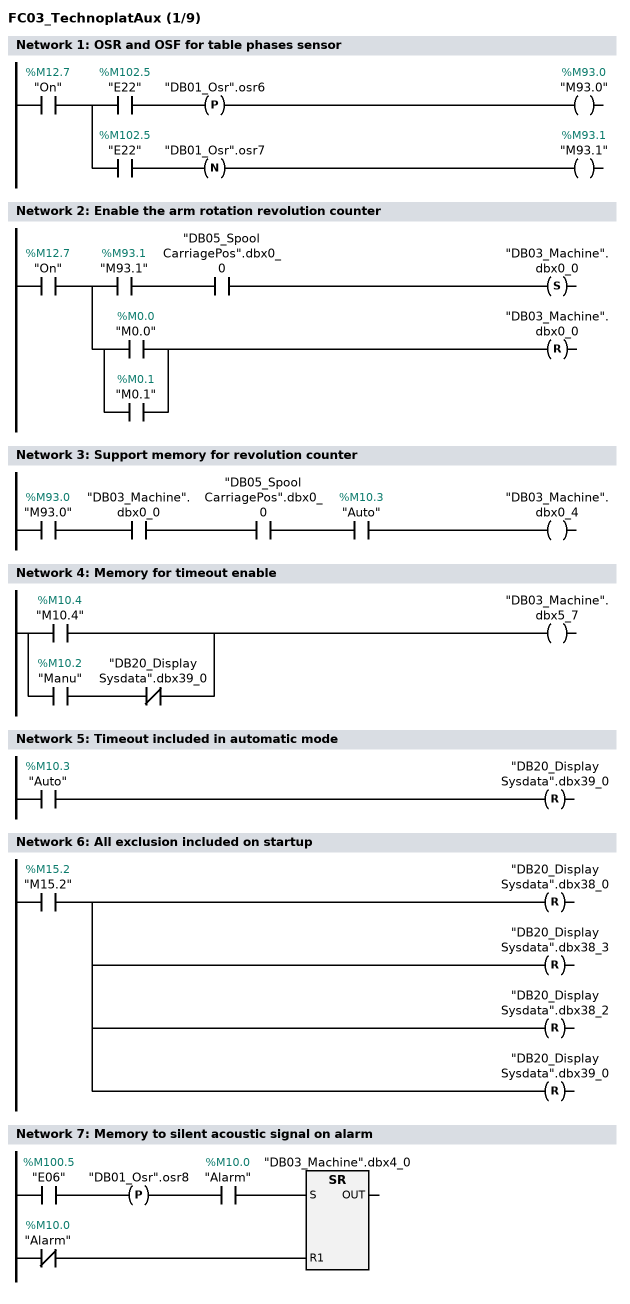
   RUNG wire#powerrail
      Contact( "On" )
      wire#w1
      Contact( "E22" )
      P_Trig( "DB01_Osr".osr6 )
      Coil( "M93.0" )
   END_RUNG
   RUNG wire#w1
      Contact( "E22" )
      N_Trig( "DB01_Osr".osr7 )
      Coil( "M93.1" )
   END_RUNG
   // the same network as SCL:
   #_w1 := "On" AND "E22";
   #_w2 := #_w1 AND NOT "DB01_Osr".osr6;   // rising edge
   "DB01_Osr".osr6 := #_w1;
   "M93.0" := #_w2;
   #_w3 := "On" AND "E22";
   #_w4 := NOT #_w3 AND "DB01_Osr".osr7;   // falling edge
   "DB01_Osr".osr7 := #_w3;
   "M93.1" := #_w4;
END_REGION

REGION Network 2: Enable the arm rotation revolution counter
   RUNG wire#powerrail
      Contact( "On" )
      wire#w1
      Contact( "M93.1" )
      Contact( "DB05_SpoolCarriagePos".dbx0_0 )
      S_Coil( "DB03_Machine".dbx0_0 )
   END_RUNG
   RUNG wire#w1
      Contact( "M0.0" )
      wire#w2
      R_Coil( "DB03_Machine".dbx0_0 )
   END_RUNG
   RUNG wire#w1
      Contact( "M0.1" )
   END_RUNG wire#w2
   // the same network as SCL:
   IF "On" AND "M93.1" AND "DB05_SpoolCarriagePos".dbx0_0 THEN "DB03_Machine".dbx0_0 := TRUE; END_IF;
   IF "On" AND ("M0.0" OR "M0.1") THEN "DB03_Machine".dbx0_0 := FALSE; END_IF;
END_REGION

REGION Network 3: Support memory for revolution counter
   RUNG wire#powerrail
      Contact( "M93.0" )
      Contact( "DB03_Machine".dbx0_0 )
      Contact( "DB05_SpoolCarriagePos".dbx0_0 )
      Contact( "Auto" )
      Coil( "DB03_Machine".dbx0_4 )
   END_RUNG
   // the same network as SCL:
   "DB03_Machine".dbx0_4 := "M93.0" AND "DB03_Machine".dbx0_0 AND "DB05_SpoolCarriagePos".dbx0_0 AND "Auto";
END_REGION

REGION Network 4: Memory for timeout enable
   RUNG wire#powerrail
      Contact( "M10.4" )
      wire#w1
      Coil( "DB03_Machine".dbx5_7 )
   END_RUNG
   RUNG wire#powerrail
      Contact( "Manu" )
      I_Contact( "DB20_DisplaySysdata".dbx39_0 )
   END_RUNG wire#w1
   // the same network as SCL:
   "DB03_Machine".dbx5_7 := "M10.4" OR ("Manu" AND NOT "DB20_DisplaySysdata".dbx39_0);
END_REGION

REGION Network 5: Timeout included in automatic mode
   RUNG wire#powerrail
      Contact( "Auto" )
      R_Coil( "DB20_DisplaySysdata".dbx39_0 )
   END_RUNG
   // the same network as SCL:
   IF "Auto" THEN "DB20_DisplaySysdata".dbx39_0 := FALSE; END_IF;
END_REGION

REGION Network 6: All exclusion included on startup
   RUNG wire#powerrail
      Contact( "M15.2" )
      wire#w1
      R_Coil( "DB20_DisplaySysdata".dbx38_0 )
   END_RUNG
   RUNG wire#w1
      R_Coil( "DB20_DisplaySysdata".dbx38_3 )
   END_RUNG
   RUNG wire#w1
      R_Coil( "DB20_DisplaySysdata".dbx38_2 )
   END_RUNG
   RUNG wire#w1
      R_Coil( "DB20_DisplaySysdata".dbx39_0 )
   END_RUNG
   // the same network as SCL:
   IF "M15.2" THEN
       "DB20_DisplaySysdata".dbx38_0 := FALSE;
       "DB20_DisplaySysdata".dbx38_3 := FALSE;
       "DB20_DisplaySysdata".dbx38_2 := FALSE;
       "DB20_DisplaySysdata".dbx39_0 := FALSE;
   END_IF;
END_REGION

REGION Network 7: Memory to silent acoustic signal on alarm
   RUNG wire#powerrail
      Contact( "E06" )
      P_Trig( "DB01_Osr".osr8 )
      Contact( "Alarm" )
      S_SR(operand := "DB03_Machine".dbx4_0, r1 := wire#w1)
   END_RUNG
   RUNG wire#powerrail
      I_Contact( "Alarm" )
   END_RUNG wire#w1
   // the same network as SCL:
   #_w1 := "E06" AND NOT "DB01_Osr".osr8;   // rising edge
   "DB01_Osr".osr8 := "E06";
   IF #_w1 AND "Alarm" THEN
       "DB03_Machine".dbx4_0 := TRUE;   // SR flip-flop
   END_IF;
   IF NOT "Alarm" THEN "DB03_Machine".dbx4_0 := FALSE; END_IF;
END_REGION

REGION Network 8: All units are ready for automatic cycle
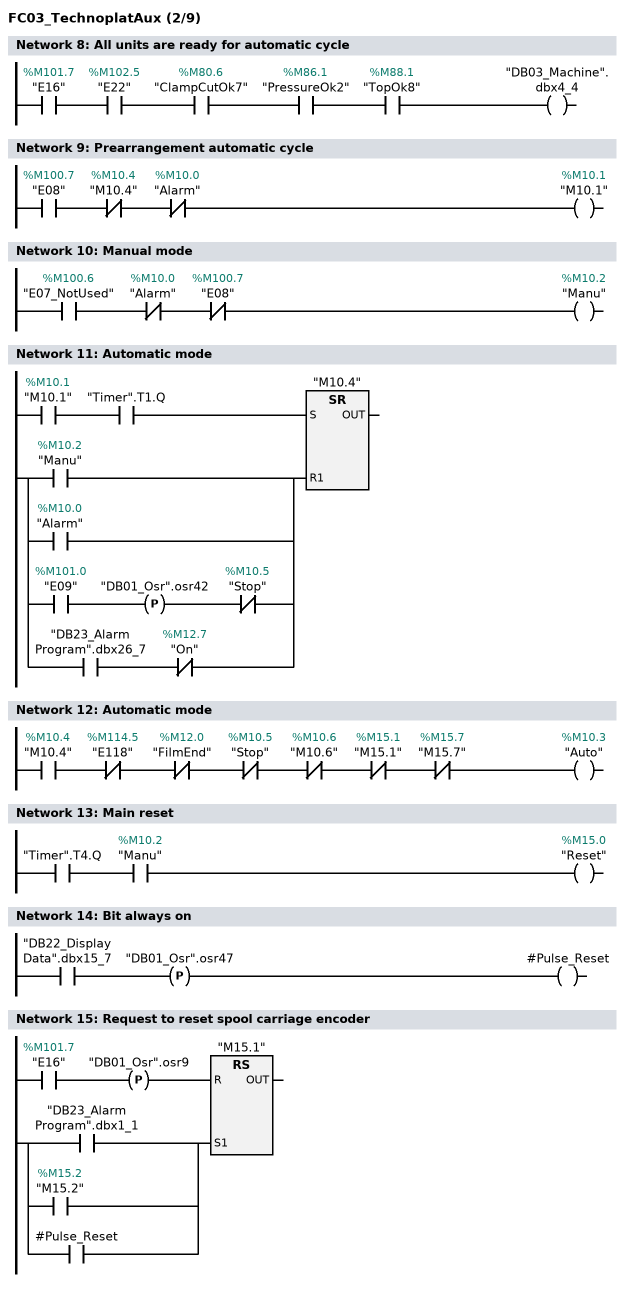
   RUNG wire#powerrail
      Contact( "E16" )
      Contact( "E22" )
      Contact( "ClampCutOk7" )
      Contact( "PressureOk2" )
      Contact( "TopOk8" )
      Coil( "DB03_Machine".dbx4_4 )
   END_RUNG
   // the same network as SCL:
   "DB03_Machine".dbx4_4 := "E16" AND "E22" AND "ClampCutOk7" AND "PressureOk2" AND "TopOk8";
END_REGION

REGION Network 9: Prearrangement automatic cycle
   RUNG wire#powerrail
      Contact( "E08" )
      I_Contact( "M10.4" )
      I_Contact( "Alarm" )
      Coil( "M10.1" )
   END_RUNG
   // the same network as SCL:
   "M10.1" := "E08" AND NOT "M10.4" AND NOT "Alarm";
END_REGION

REGION Network 10: Manual mode
   RUNG wire#powerrail
      Contact( "E07_NotUsed" )
      I_Contact( "Alarm" )
      I_Contact( "E08" )
      Coil( "Manu" )
   END_RUNG
   // the same network as SCL:
   "Manu" := "E07_NotUsed" AND NOT "Alarm" AND NOT "E08";
END_REGION

REGION Network 11: Automatic mode
   RUNG wire#powerrail
      Contact( "M10.1" )
      Contact( "Timer".T1.Q )
      S_SR(operand := "M10.4", r1 := wire#w1)
   END_RUNG
   RUNG wire#powerrail
      Contact( "Manu" )
   END_RUNG wire#w1
   RUNG wire#powerrail
      Contact( "Alarm" )
   END_RUNG wire#w1
   RUNG wire#powerrail
      Contact( "E09" )
      P_Trig( "DB01_Osr".osr42 )
      I_Contact( "Stop" )
   END_RUNG wire#w1
   RUNG wire#powerrail
      Contact( "DB23_AlarmProgram".dbx26_7 )
      I_Contact( "On" )
   END_RUNG wire#w1
   // the same network as SCL:
   #_w1 := "E09" AND NOT "DB01_Osr".osr42;   // rising edge
   "DB01_Osr".osr42 := "E09";
   IF "M10.1" AND "Timer".T1.Q THEN
       "M10.4" := TRUE;   // SR flip-flop
   END_IF;
   IF "Manu" OR "Alarm" OR (#_w1 AND NOT "Stop") OR ("DB23_AlarmProgram".dbx26_7 AND NOT "On") THEN
       "M10.4" := FALSE;
   END_IF;
END_REGION

REGION Network 12: Automatic mode
   RUNG wire#powerrail
      Contact( "M10.4" )
      I_Contact( "E118" )
      I_Contact( "FilmEnd" )
      I_Contact( "Stop" )
      I_Contact( "M10.6" )
      I_Contact( "M15.1" )
      I_Contact( "M15.7" )
      Coil( "Auto" )
   END_RUNG
   // the same network as SCL:
   "Auto" := "M10.4" AND NOT "E118" AND NOT "FilmEnd" AND NOT "Stop" AND NOT "M10.6" AND NOT "M15.1" AND NOT "M15.7";
END_REGION

REGION Network 13: Main reset
   RUNG wire#powerrail
      Contact( "Timer".T4.Q )
      Contact( "Manu" )
      Coil( "Reset" )
   END_RUNG
   // the same network as SCL:
   "Reset" := "Timer".T4.Q AND "Manu";
END_REGION

REGION Network 14: Bit always on
   RUNG wire#powerrail
      Contact( "DB22_DisplayData".dbx15_7 )
      P_Trig( "DB01_Osr".osr47 )
      Coil( #Pulse_Reset )
   END_RUNG
   // the same network as SCL:
   #_w1 := "DB22_DisplayData".dbx15_7 AND NOT "DB01_Osr".osr47;   // rising edge
   "DB01_Osr".osr47 := "DB22_DisplayData".dbx15_7;
   #Pulse_Reset := #_w1;
END_REGION

REGION Network 15: Request to reset spool carriage encoder
   RUNG wire#powerrail
      Contact( "E16" )
      P_Trig( "DB01_Osr".osr9 )
      S_RS(operand := "M15.1", s1 := wire#w1)
   END_RUNG
   RUNG wire#powerrail
      Contact( "DB23_AlarmProgram".dbx1_1 )
   END_RUNG wire#w1
   RUNG wire#powerrail
      Contact( "M15.2" )
   END_RUNG wire#w1
   RUNG wire#powerrail
      Contact( #Pulse_Reset )
   END_RUNG wire#w1
   // the same network as SCL:
   #_w1 := "E16" AND NOT "DB01_Osr".osr9;   // rising edge
   "DB01_Osr".osr9 := "E16";
   IF #_w1 THEN
       "M15.1" := FALSE;   // RS flip-flop
   END_IF;
   IF "DB23_AlarmProgram".dbx1_1 OR "M15.2" OR #Pulse_Reset THEN "M15.1" := TRUE; END_IF;
END_REGION

REGION Network 16: Request to reset table rotation encoder
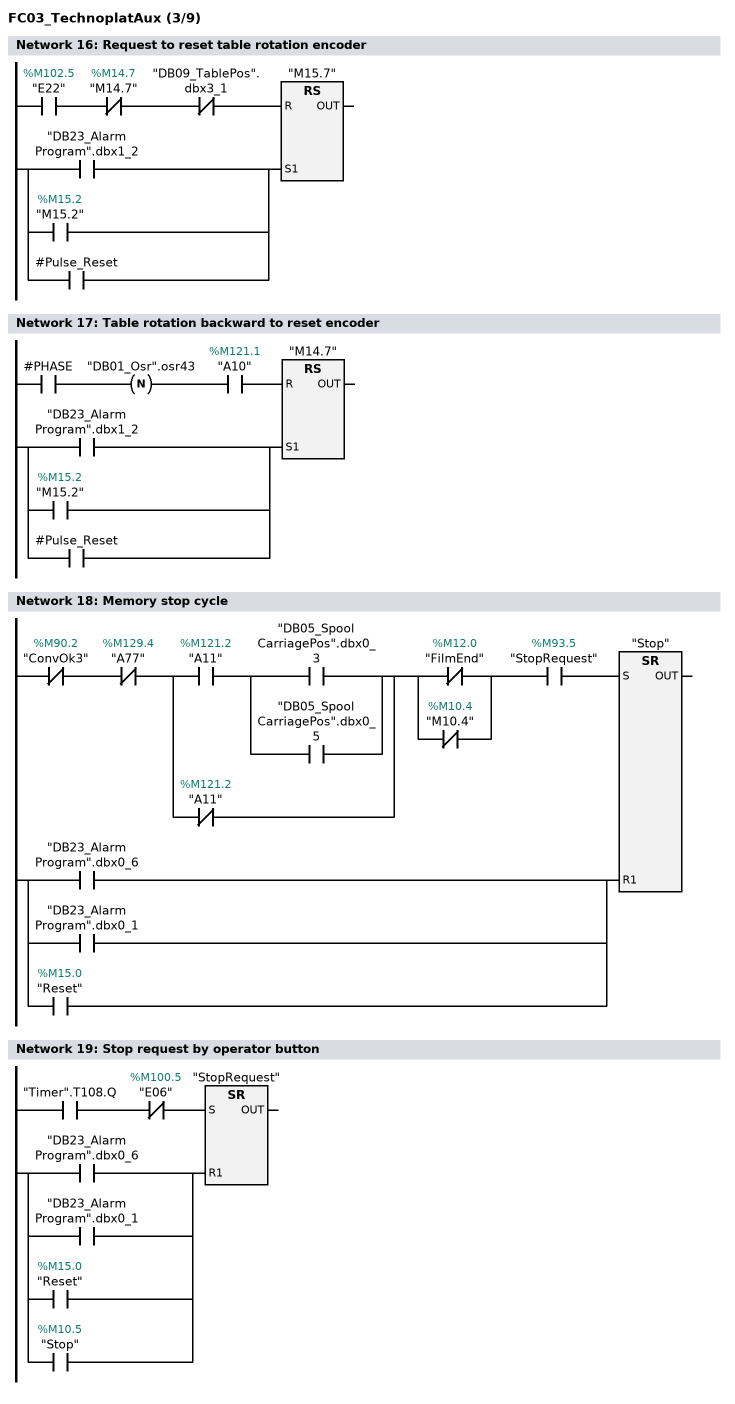
   RUNG wire#powerrail
      Contact( "E22" )
      I_Contact( "M14.7" )
      I_Contact( "DB09_TablePos".dbx3_1 )
      S_RS(operand := "M15.7", s1 := wire#w1)
   END_RUNG
   RUNG wire#powerrail
      Contact( "DB23_AlarmProgram".dbx1_2 )
   END_RUNG wire#w1
   RUNG wire#powerrail
      Contact( "M15.2" )
   END_RUNG wire#w1
   RUNG wire#powerrail
      Contact( #Pulse_Reset )
   END_RUNG wire#w1
   // the same network as SCL:
   IF "E22" AND NOT "M14.7" AND NOT "DB09_TablePos".dbx3_1 THEN
       "M15.7" := FALSE;   // RS flip-flop
   END_IF;
   IF "DB23_AlarmProgram".dbx1_2 OR "M15.2" OR #Pulse_Reset THEN "M15.7" := TRUE; END_IF;
END_REGION

REGION Network 17: Table rotation backward to reset encoder
   RUNG wire#powerrail
      Contact( #PHASE )
      N_Trig( "DB01_Osr".osr43 )
      Contact( "A10" )
      S_RS(operand := "M14.7", s1 := wire#w1)
   END_RUNG
   RUNG wire#powerrail
      Contact( "DB23_AlarmProgram".dbx1_2 )
   END_RUNG wire#w1
   RUNG wire#powerrail
      Contact( "M15.2" )
   END_RUNG wire#w1
   RUNG wire#powerrail
      Contact( #Pulse_Reset )
   END_RUNG wire#w1
   // the same network as SCL:
   #_w1 := NOT #PHASE AND "DB01_Osr".osr43;   // falling edge
   "DB01_Osr".osr43 := #PHASE;
   IF #_w1 AND "A10" THEN
       "M14.7" := FALSE;   // RS flip-flop
   END_IF;
   IF "DB23_AlarmProgram".dbx1_2 OR "M15.2" OR #Pulse_Reset THEN "M14.7" := TRUE; END_IF;
END_REGION

REGION Network 18: Memory stop cycle
   RUNG wire#powerrail
      I_Contact( "ConvOk3" )
      I_Contact( "A77" )
      wire#w1
      Contact( "A11" )
      wire#w2
      Contact( "DB05_SpoolCarriagePos".dbx0_3 )
      wire#w3
      I_Contact( "FilmEnd" )
      wire#w4
      Contact( "StopRequest" )
      S_SR(operand := "Stop", r1 := wire#w5)
   END_RUNG
   RUNG wire#w2
      Contact( "DB05_SpoolCarriagePos".dbx0_5 )
   END_RUNG wire#w3
   RUNG wire#w1
      I_Contact( "A11" )
   END_RUNG wire#w3
   RUNG wire#w3
      I_Contact( "M10.4" )
   END_RUNG wire#w4
   RUNG wire#powerrail
      Contact( "DB23_AlarmProgram".dbx0_6 )
   END_RUNG wire#w5
   RUNG wire#powerrail
      Contact( "DB23_AlarmProgram".dbx0_1 )
   END_RUNG wire#w5
   RUNG wire#powerrail
      Contact( "Reset" )
   END_RUNG wire#w5
   // the same network as SCL:
   IF NOT "ConvOk3" AND NOT "A77" AND (("A11" AND ("DB05_SpoolCarriagePos".dbx0_3 OR "DB05_SpoolCarriagePos".dbx0_5)) OR NOT "A11") AND (NOT "FilmEnd" OR NOT "M10.4") AND "StopRequest" THEN
       "Stop" := TRUE;   // SR flip-flop
   END_IF;
   IF "DB23_AlarmProgram".dbx0_6 OR "DB23_AlarmProgram".dbx0_1 OR "Reset" THEN "Stop" := FALSE; END_IF;
END_REGION

REGION Network 19: Stop request by operator button
   RUNG wire#powerrail
      Contact( "Timer".T108.Q )
      I_Contact( "E06" )
      S_SR(operand := "StopRequest", r1 := wire#w1)
   END_RUNG
   RUNG wire#powerrail
      Contact( "DB23_AlarmProgram".dbx0_6 )
   END_RUNG wire#w1
   RUNG wire#powerrail
      Contact( "DB23_AlarmProgram".dbx0_1 )
   END_RUNG wire#w1
   RUNG wire#powerrail
      Contact( "Reset" )
   END_RUNG wire#w1
   RUNG wire#powerrail
      Contact( "Stop" )
   END_RUNG wire#w1
   // the same network as SCL:
   IF "Timer".T108.Q AND NOT "E06" THEN
       "StopRequest" := TRUE;   // SR flip-flop
   END_IF;
   IF "DB23_AlarmProgram".dbx0_6 OR "DB23_AlarmProgram".dbx0_1 OR "Reset" OR "Stop" THEN
       "StopRequest" := FALSE;
   END_IF;
END_REGION

REGION Network 20: Memory to stop cycle for door open request
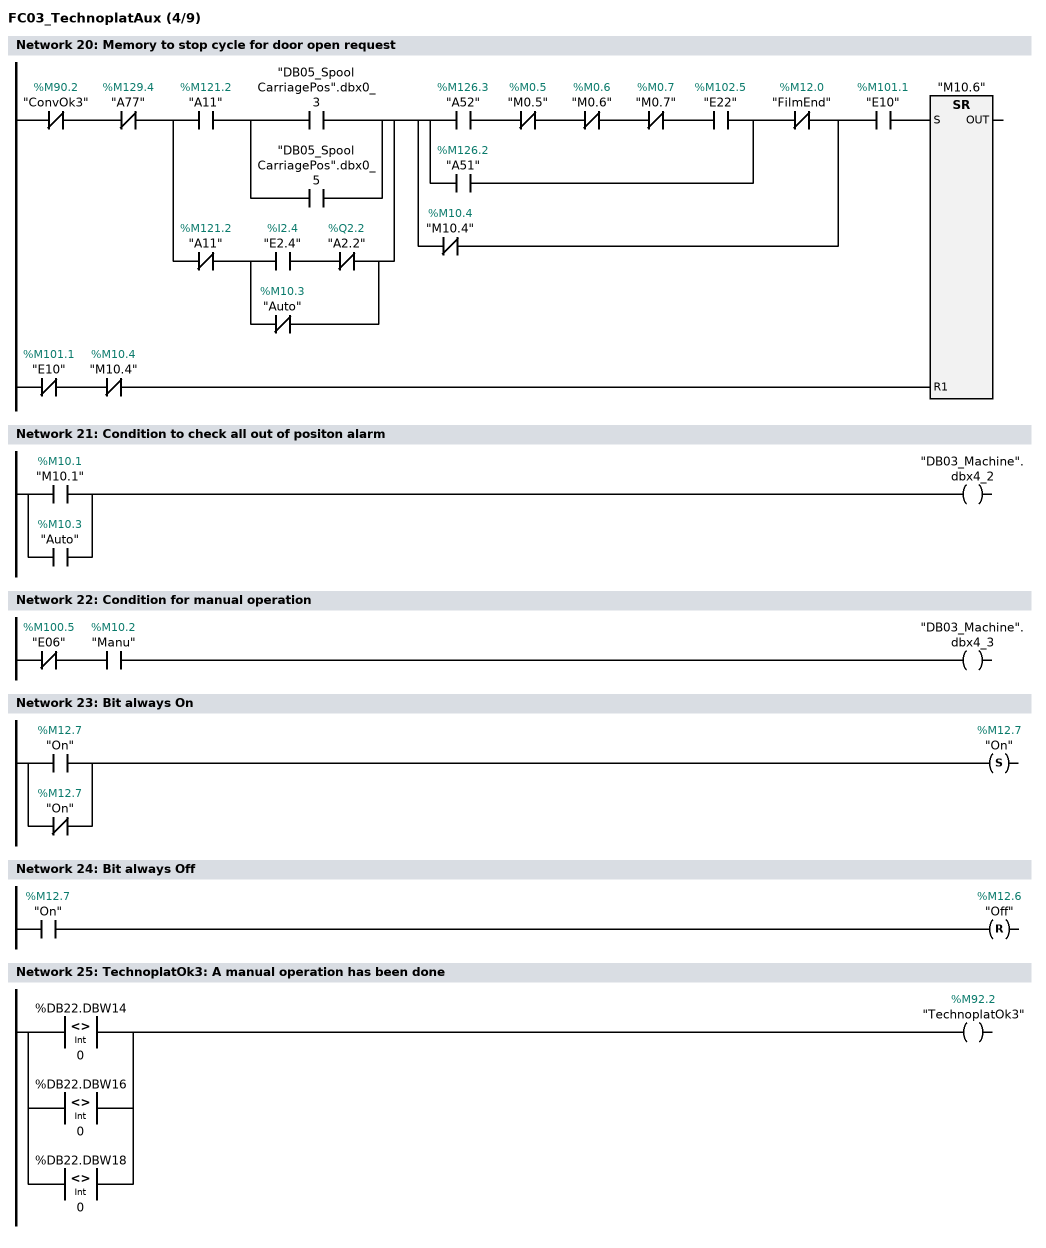
   RUNG wire#powerrail
      I_Contact( "ConvOk3" )
      I_Contact( "A77" )
      wire#w1
      Contact( "A11" )
      wire#w2
      Contact( "DB05_SpoolCarriagePos".dbx0_3 )
      wire#w3
      Contact( "A52" )
      I_Contact( "M0.5" )
      I_Contact( "M0.6" )
      I_Contact( "M0.7" )
      Contact( "E22" )
      wire#w5
      I_Contact( "FilmEnd" )
      wire#w6
      Contact( "E10" )
      S_SR(operand := "M10.6", r1 := wire#w7)
   END_RUNG
   RUNG wire#w2
      Contact( "DB05_SpoolCarriagePos".dbx0_5 )
   END_RUNG wire#w3
   RUNG wire#w1
      I_Contact( "A11" )
      wire#w4
      Contact( "E2.4" )
      I_Contact( "A2.2" )
   END_RUNG wire#w3
   RUNG wire#w4
      I_Contact( "Auto" )
   END_RUNG wire#w3
   RUNG wire#w3
      Contact( "A51" )
   END_RUNG wire#w5
   RUNG wire#w3
      I_Contact( "M10.4" )
   END_RUNG wire#w6
   RUNG wire#powerrail
      I_Contact( "E10" )
      I_Contact( "M10.4" )
   END_RUNG wire#w7
   // the same network as SCL:
   IF NOT "ConvOk3" AND NOT "A77" AND (("A11" AND ("DB05_SpoolCarriagePos".dbx0_3 OR "DB05_SpoolCarriagePos".dbx0_5)) OR (NOT "A11" AND (("E2.4" AND NOT "A2.2") OR NOT "Auto"))) AND (((("A52" AND NOT "M0.5" AND NOT "M0.6" AND NOT "M0.7" AND "E22") OR "A51") AND NOT "FilmEnd") OR NOT "M10.4") AND "E10" THEN
       "M10.6" := TRUE;   // SR flip-flop
   END_IF;
   IF NOT "E10" AND NOT "M10.4" THEN "M10.6" := FALSE; END_IF;
END_REGION

REGION Network 21: Condition to check all out of positon alarm
   RUNG wire#powerrail
      Contact( "M10.1" )
      wire#w1
      Coil( "DB03_Machine".dbx4_2 )
   END_RUNG
   RUNG wire#powerrail
      Contact( "Auto" )
   END_RUNG wire#w1
   // the same network as SCL:
   "DB03_Machine".dbx4_2 := "M10.1" OR "Auto";
END_REGION

REGION Network 22: Condition for manual operation
   RUNG wire#powerrail
      I_Contact( "E06" )
      Contact( "Manu" )
      Coil( "DB03_Machine".dbx4_3 )
   END_RUNG
   // the same network as SCL:
   "DB03_Machine".dbx4_3 := NOT "E06" AND "Manu";
END_REGION

REGION Network 23: Bit always On
   RUNG wire#powerrail
      Contact( "On" )
      wire#w1
      S_Coil( "On" )
   END_RUNG
   RUNG wire#powerrail
      I_Contact( "On" )
   END_RUNG wire#w1
   // the same network as SCL:
   IF "On" OR NOT "On" THEN "On" := TRUE; END_IF;
END_REGION

REGION Network 24: Bit always Off
   RUNG wire#powerrail
      Contact( "On" )
      R_Coil( "Off" )
   END_RUNG
   // the same network as SCL:
   IF "On" THEN "Off" := FALSE; END_IF;
END_REGION

REGION Network 25: TechnoplatOk3: A manual operation has been done
   RUNG wire#powerrail
      { S7_Templates := "SrcType := Int" } NE_Contact(in1 := %DB22.DBW14, in2 := 0)
      wire#w1
      Coil( "TechnoplatOk3" )
   END_RUNG
   RUNG wire#powerrail
      { S7_Templates := "SrcType := Int" } NE_Contact(in1 := %DB22.DBW16, in2 := 0)
   END_RUNG wire#w1
   RUNG wire#powerrail
      { S7_Templates := "SrcType := Int" } NE_Contact(in1 := %DB22.DBW18, in2 := 0)
   END_RUNG wire#w1
   // the same network as SCL:
   "TechnoplatOk3" := (%DB22.DBW14 <> 0) OR (%DB22.DBW16 <> 0) OR (%DB22.DBW18 <> 0);
END_REGION

REGION Network 26: Alarm - Warning reset
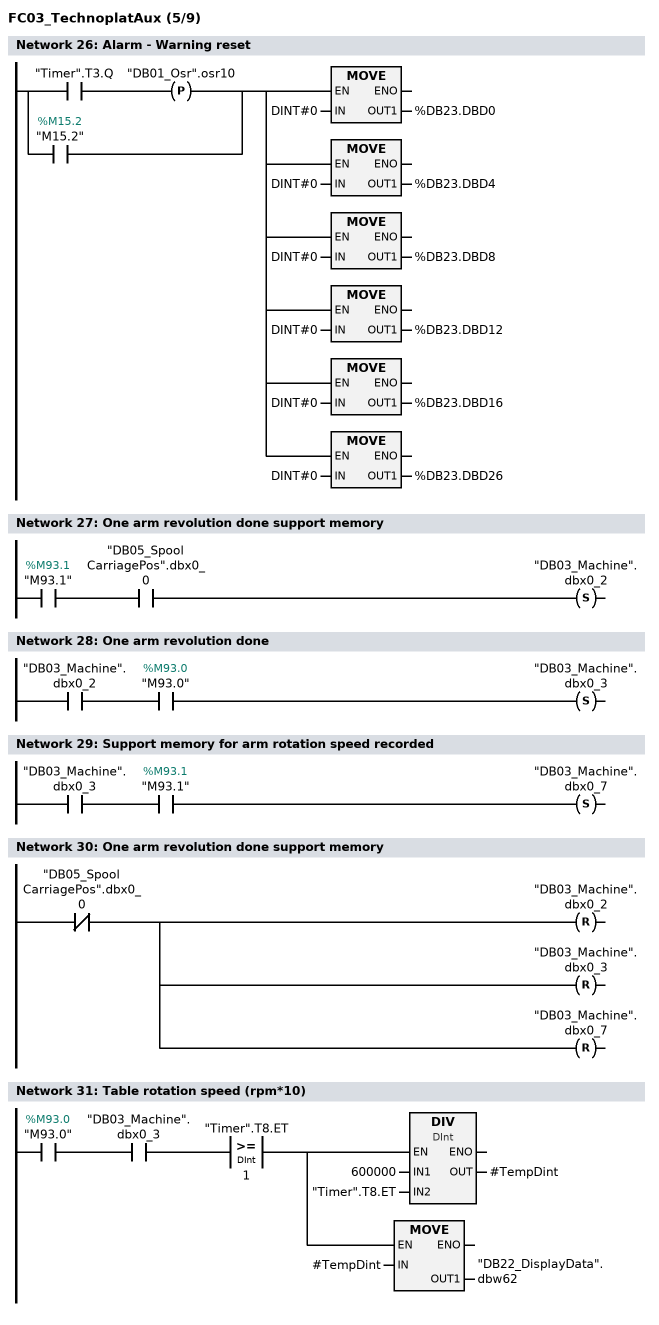
   RUNG wire#powerrail
      Contact( "Timer".T3.Q )
      P_Trig( "DB01_Osr".osr10 )
      wire#w1
      { S7_GenerateENO := "TRUE" } Move(in := DINT#0, out1 => %DB23.DBD0)
   END_RUNG
   RUNG wire#powerrail
      Contact( "M15.2" )
   END_RUNG wire#w1
   RUNG wire#w1
      { S7_GenerateENO := "TRUE" } Move(in := DINT#0, out1 => %DB23.DBD4)
   END_RUNG
   RUNG wire#w1
      { S7_GenerateENO := "TRUE" } Move(in := DINT#0, out1 => %DB23.DBD8)
   END_RUNG
   RUNG wire#w1
      { S7_GenerateENO := "TRUE" } Move(in := DINT#0, out1 => %DB23.DBD12)
   END_RUNG
   RUNG wire#w1
      { S7_GenerateENO := "TRUE" } Move(in := DINT#0, out1 => %DB23.DBD16)
   END_RUNG
   RUNG wire#w1
      { S7_GenerateENO := "TRUE" } Move(in := DINT#0, out1 => %DB23.DBD26)
   END_RUNG
   // the same network as SCL:
   #_w1 := "Timer".T3.Q AND NOT "DB01_Osr".osr10;   // rising edge
   "DB01_Osr".osr10 := "Timer".T3.Q;
   IF #_w1 OR "M15.2" THEN
       %DB23.DBD0 := DINT#0;
       %DB23.DBD4 := DINT#0;
       %DB23.DBD8 := DINT#0;
       %DB23.DBD12 := DINT#0;
       %DB23.DBD16 := DINT#0;
       %DB23.DBD26 := DINT#0;
   END_IF;
END_REGION

REGION Network 27: One arm revolution done support memory
   RUNG wire#powerrail
      Contact( "M93.1" )
      Contact( "DB05_SpoolCarriagePos".dbx0_0 )
      S_Coil( "DB03_Machine".dbx0_2 )
   END_RUNG
   // the same network as SCL:
   IF "M93.1" AND "DB05_SpoolCarriagePos".dbx0_0 THEN "DB03_Machine".dbx0_2 := TRUE; END_IF;
END_REGION

REGION Network 28: One arm revolution done
   RUNG wire#powerrail
      Contact( "DB03_Machine".dbx0_2 )
      Contact( "M93.0" )
      S_Coil( "DB03_Machine".dbx0_3 )
   END_RUNG
   // the same network as SCL:
   IF "DB03_Machine".dbx0_2 AND "M93.0" THEN "DB03_Machine".dbx0_3 := TRUE; END_IF;
END_REGION

REGION Network 29: Support memory for arm rotation speed recorded
   RUNG wire#powerrail
      Contact( "DB03_Machine".dbx0_3 )
      Contact( "M93.1" )
      S_Coil( "DB03_Machine".dbx0_7 )
   END_RUNG
   // the same network as SCL:
   IF "DB03_Machine".dbx0_3 AND "M93.1" THEN "DB03_Machine".dbx0_7 := TRUE; END_IF;
END_REGION

REGION Network 30: One arm revolution done support memory
   RUNG wire#powerrail
      I_Contact( "DB05_SpoolCarriagePos".dbx0_0 )
      wire#w1
      R_Coil( "DB03_Machine".dbx0_2 )
   END_RUNG
   RUNG wire#w1
      R_Coil( "DB03_Machine".dbx0_3 )
   END_RUNG
   RUNG wire#w1
      R_Coil( "DB03_Machine".dbx0_7 )
   END_RUNG
   // the same network as SCL:
   IF NOT "DB05_SpoolCarriagePos".dbx0_0 THEN
       "DB03_Machine".dbx0_2 := FALSE;
       "DB03_Machine".dbx0_3 := FALSE;
       "DB03_Machine".dbx0_7 := FALSE;
   END_IF;
END_REGION

REGION Network 31: Table rotation speed (rpm*10)
   RUNG wire#powerrail
      Contact( "M93.0" )
      Contact( "DB03_Machine".dbx0_3 )
      { S7_Templates := "SrcType := DInt" } GE_Contact(in1 := "Timer".T8.ET, in2 := 1)
      wire#w1
      { S7_Templates := "SrcType := DInt"; S7_GenerateENO := "TRUE" } Div(in1 := 600000, in2 := "Timer".T8.ET, out => #TempDint)
   END_RUNG
   RUNG wire#w1
      { S7_GenerateENO := "TRUE" } Move(in := #TempDint, out1 => "DB22_DisplayData".dbw62)
   END_RUNG
   // the same network as SCL:
   IF "M93.0" AND "DB03_Machine".dbx0_3 AND ("Timer".T8.ET >= 1) THEN
       #TempDint := 600000 / "Timer".T8.ET;
       "DB22_DisplayData".dbw62 := #TempDint;
   END_IF;
END_REGION

REGION Network 32: Arm rotation speed
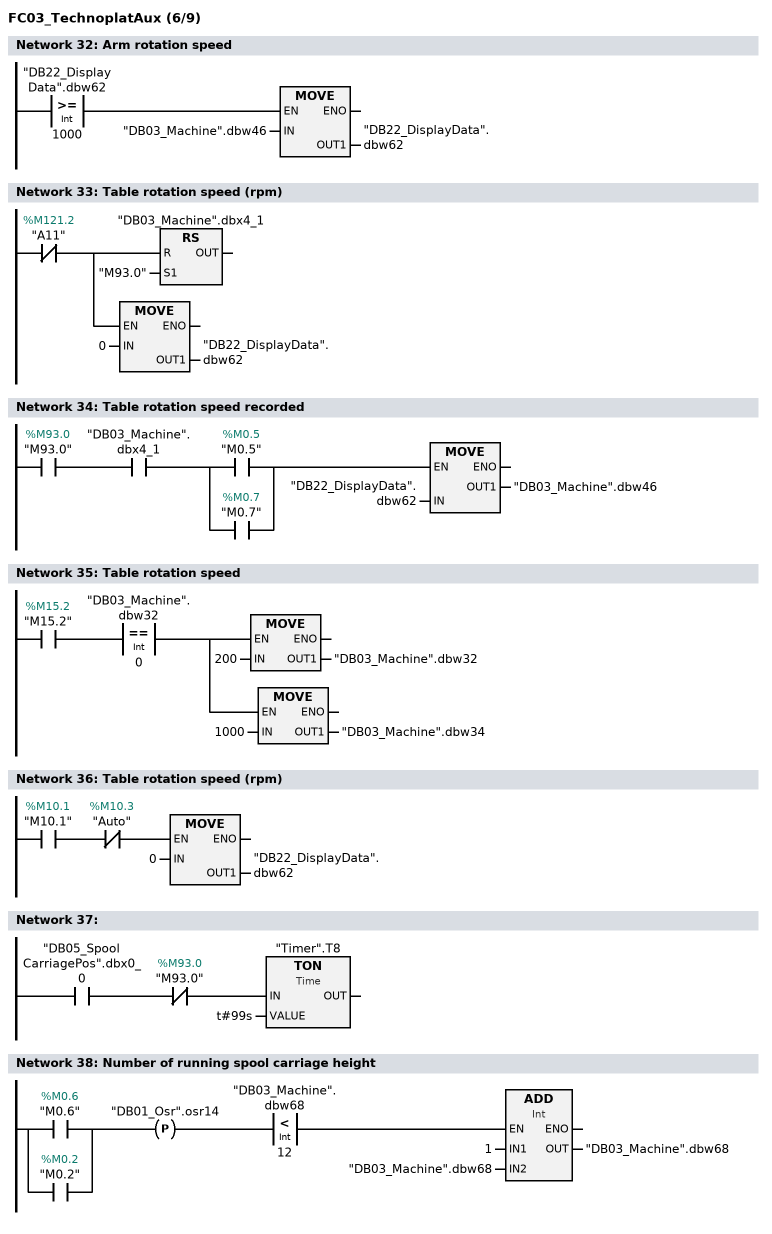
   RUNG wire#powerrail
      { S7_Templates := "SrcType := Int" } GE_Contact(in1 := "DB22_DisplayData".dbw62, in2 := 1000)
      { S7_GenerateENO := "TRUE" } Move(in := "DB03_Machine".dbw46, out1 => "DB22_DisplayData".dbw62)
   END_RUNG
   // the same network as SCL:
   IF "DB22_DisplayData".dbw62 >= 1000 THEN "DB22_DisplayData".dbw62 := "DB03_Machine".dbw46; END_IF;
END_REGION

REGION Network 33: Table rotation speed (rpm)
   RUNG wire#powerrail
      I_Contact( "A11" )
      wire#w1
      S_RS(operand := "DB03_Machine".dbx4_1, s1 := "M93.0")
   END_RUNG
   RUNG wire#w1
      { S7_GenerateENO := "TRUE" } Move(in := 0, out1 => "DB22_DisplayData".dbw62)
   END_RUNG
   // the same network as SCL:
   IF NOT "A11" THEN
       "DB03_Machine".dbx4_1 := FALSE;   // RS flip-flop
   END_IF;
   IF "M93.0" THEN "DB03_Machine".dbx4_1 := TRUE; END_IF;
   IF NOT "A11" THEN "DB22_DisplayData".dbw62 := 0; END_IF;
END_REGION

REGION Network 34: Table rotation speed recorded
   RUNG wire#powerrail
      Contact( "M93.0" )
      Contact( "DB03_Machine".dbx4_1 )
      wire#w1
      Contact( "M0.5" )
      wire#w2
      { S7_GenerateENO := "TRUE" } Move(in := "DB22_DisplayData".dbw62, out1 => "DB03_Machine".dbw46)
   END_RUNG
   RUNG wire#w1
      Contact( "M0.7" )
   END_RUNG wire#w2
   // the same network as SCL:
   IF "M93.0" AND "DB03_Machine".dbx4_1 AND ("M0.5" OR "M0.7") THEN
       "DB03_Machine".dbw46 := "DB22_DisplayData".dbw62;
   END_IF;
END_REGION

REGION Network 35: Table rotation speed
   RUNG wire#powerrail
      Contact( "M15.2" )
      { S7_Templates := "SrcType := Int" } EQ_Contact(in1 := "DB03_Machine".dbw32, in2 := 0)
      wire#w1
      { S7_GenerateENO := "TRUE" } Move(in := 200, out1 => "DB03_Machine".dbw32)
   END_RUNG
   RUNG wire#w1
      { S7_GenerateENO := "TRUE" } Move(in := 1000, out1 => "DB03_Machine".dbw34)
   END_RUNG
   // the same network as SCL:
   #_w1 := "M15.2" AND ("DB03_Machine".dbw32 = 0);
   IF #_w1 THEN
       "DB03_Machine".dbw32 := 200;
       "DB03_Machine".dbw34 := 1000;
   END_IF;
END_REGION

REGION Network 36: Table rotation speed (rpm)
   RUNG wire#powerrail
      Contact( "M10.1" )
      I_Contact( "Auto" )
      { S7_GenerateENO := "TRUE" } Move(in := 0, out1 => "DB22_DisplayData".dbw62)
   END_RUNG
   // the same network as SCL:
   IF "M10.1" AND NOT "Auto" THEN "DB22_DisplayData".dbw62 := 0; END_IF;
END_REGION

REGION Network 37
   "Timer".T8.TON(IN := "DB05_SpoolCarriagePos".dbx0_0 AND NOT "M93.0", PT := t#99s);   // TON coil
END_REGION

REGION Network 38: Number of running spool carriage height
   RUNG wire#powerrail
      Contact( "M0.6" )
      wire#w1
      P_Trig( "DB01_Osr".osr14 )
      { S7_Templates := "SrcType := Int" } LT_Contact(in1 := "DB03_Machine".dbw68, in2 := 12)
      { S7_Templates := "SrcType := Int"; S7_GenerateENO := "TRUE" } Add(in1 := 1, in2 := "DB03_Machine".dbw68, out => "DB03_Machine".dbw68)
   END_RUNG
   RUNG wire#powerrail
      Contact( "M0.2" )
   END_RUNG wire#w1
   // the same network as SCL:
   #_w1 := "M0.6" OR "M0.2";
   #_w2 := #_w1 AND NOT "DB01_Osr".osr14;   // rising edge
   "DB01_Osr".osr14 := #_w1;
   IF #_w2 AND ("DB03_Machine".dbw68 < 12) THEN "DB03_Machine".dbw68 := 1 + "DB03_Machine".dbw68; END_IF;
END_REGION

REGION Network 39: Number of running spool carriage height
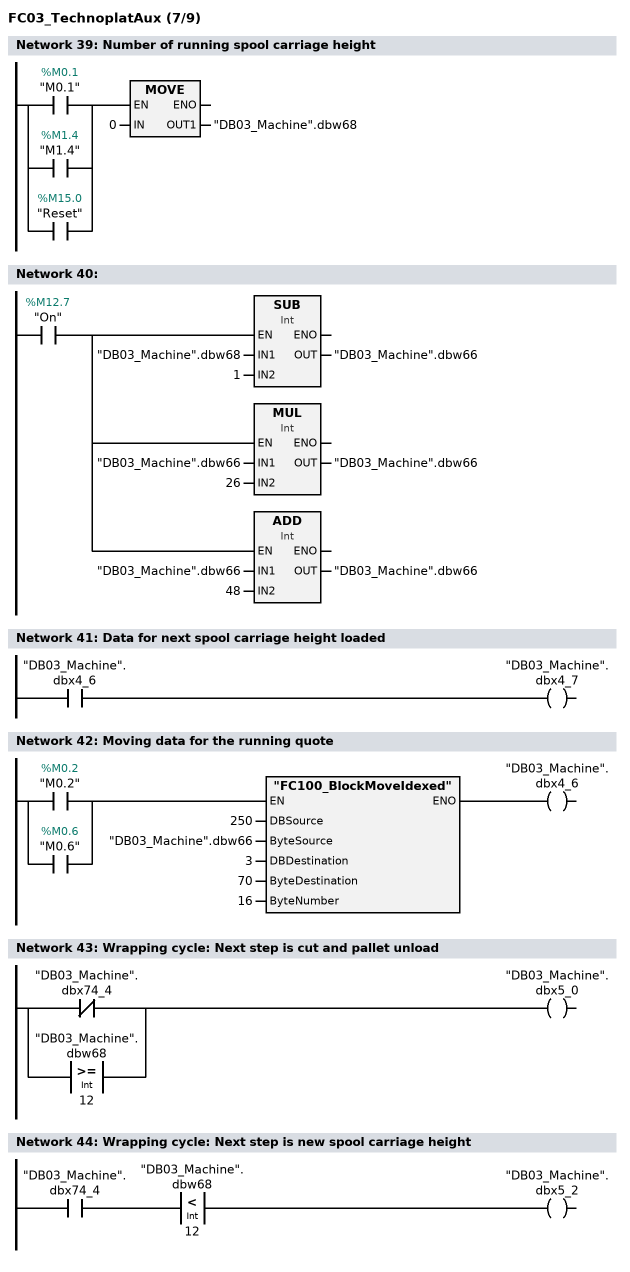
   RUNG wire#powerrail
      Contact( "M0.1" )
      wire#w1
      { S7_GenerateENO := "TRUE" } Move(in := 0, out1 => "DB03_Machine".dbw68)
   END_RUNG
   RUNG wire#powerrail
      Contact( "M1.4" )
   END_RUNG wire#w1
   RUNG wire#powerrail
      Contact( "Reset" )
   END_RUNG wire#w1
   // the same network as SCL:
   IF "M0.1" OR "M1.4" OR "Reset" THEN "DB03_Machine".dbw68 := 0; END_IF;
END_REGION

REGION Network 40
   RUNG wire#powerrail
      Contact( "On" )
      wire#w1
      { S7_Templates := "SrcType := Int"; S7_GenerateENO := "TRUE" } Sub(in1 := "DB03_Machine".dbw68, in2 := 1, out => "DB03_Machine".dbw66)
   END_RUNG
   RUNG wire#w1
      { S7_Templates := "SrcType := Int"; S7_GenerateENO := "TRUE" } Mul(in1 := "DB03_Machine".dbw66, in2 := 26, out => "DB03_Machine".dbw66)
   END_RUNG
   RUNG wire#w1
      { S7_Templates := "SrcType := Int"; S7_GenerateENO := "TRUE" } Add(in1 := "DB03_Machine".dbw66, in2 := 48, out => "DB03_Machine".dbw66)
   END_RUNG
   // the same network as SCL:
   IF "On" THEN
       "DB03_Machine".dbw66 := "DB03_Machine".dbw68 - 1;
       "DB03_Machine".dbw66 := "DB03_Machine".dbw66 * 26;
       "DB03_Machine".dbw66 := "DB03_Machine".dbw66 + 48;
   END_IF;
END_REGION

REGION Network 41: Data for next spool carriage height loaded
   RUNG wire#powerrail
      Contact( "DB03_Machine".dbx4_6 )
      Coil( "DB03_Machine".dbx4_7 )
   END_RUNG
   // the same network as SCL:
   "DB03_Machine".dbx4_7 := "DB03_Machine".dbx4_6;
END_REGION

REGION Network 42: Moving data for the running quote
   RUNG wire#powerrail
      Contact( "M0.2" )
      wire#w1
      "FC100_BlockMoveIdexed"(DBSource := 250, ByteSource := "DB03_Machine".dbw66, DBDestination := 3, ByteDestination := 70, ByteNumber := 16)
      Coil( "DB03_Machine".dbx4_6 )
   END_RUNG
   RUNG wire#powerrail
      Contact( "M0.6" )
   END_RUNG wire#w1
   // the same network as SCL:
   "FC100_BlockMoveIdexed"(EN := "M0.2" OR "M0.6",
                           DBSource := 250,
                           ByteSource := "DB03_Machine".dbw66,
                           DBDestination := 3,
                           ByteDestination := 70,
                           ByteNumber := 16,
                           ENO => #_w1);
   "DB03_Machine".dbx4_6 := #_w1;
END_REGION

REGION Network 43: Wrapping cycle: Next step is cut and pallet unload
   RUNG wire#powerrail
      I_Contact( "DB03_Machine".dbx74_4 )
      wire#w1
      Coil( "DB03_Machine".dbx5_0 )
   END_RUNG
   RUNG wire#powerrail
      { S7_Templates := "SrcType := Int" } GE_Contact(in1 := "DB03_Machine".dbw68, in2 := 12)
   END_RUNG wire#w1
   // the same network as SCL:
   "DB03_Machine".dbx5_0 := NOT "DB03_Machine".dbx74_4 OR ("DB03_Machine".dbw68 >= 12);
END_REGION

REGION Network 44: Wrapping cycle: Next step is new spool carriage height
   RUNG wire#powerrail
      Contact( "DB03_Machine".dbx74_4 )
      { S7_Templates := "SrcType := Int" } LT_Contact(in1 := "DB03_Machine".dbw68, in2 := 12)
      Coil( "DB03_Machine".dbx5_2 )
   END_RUNG
   // the same network as SCL:
   "DB03_Machine".dbx5_2 := "DB03_Machine".dbx74_4 AND ("DB03_Machine".dbw68 < 12);
END_REGION

REGION Network 45: Wrong data program for the pallet on the machine
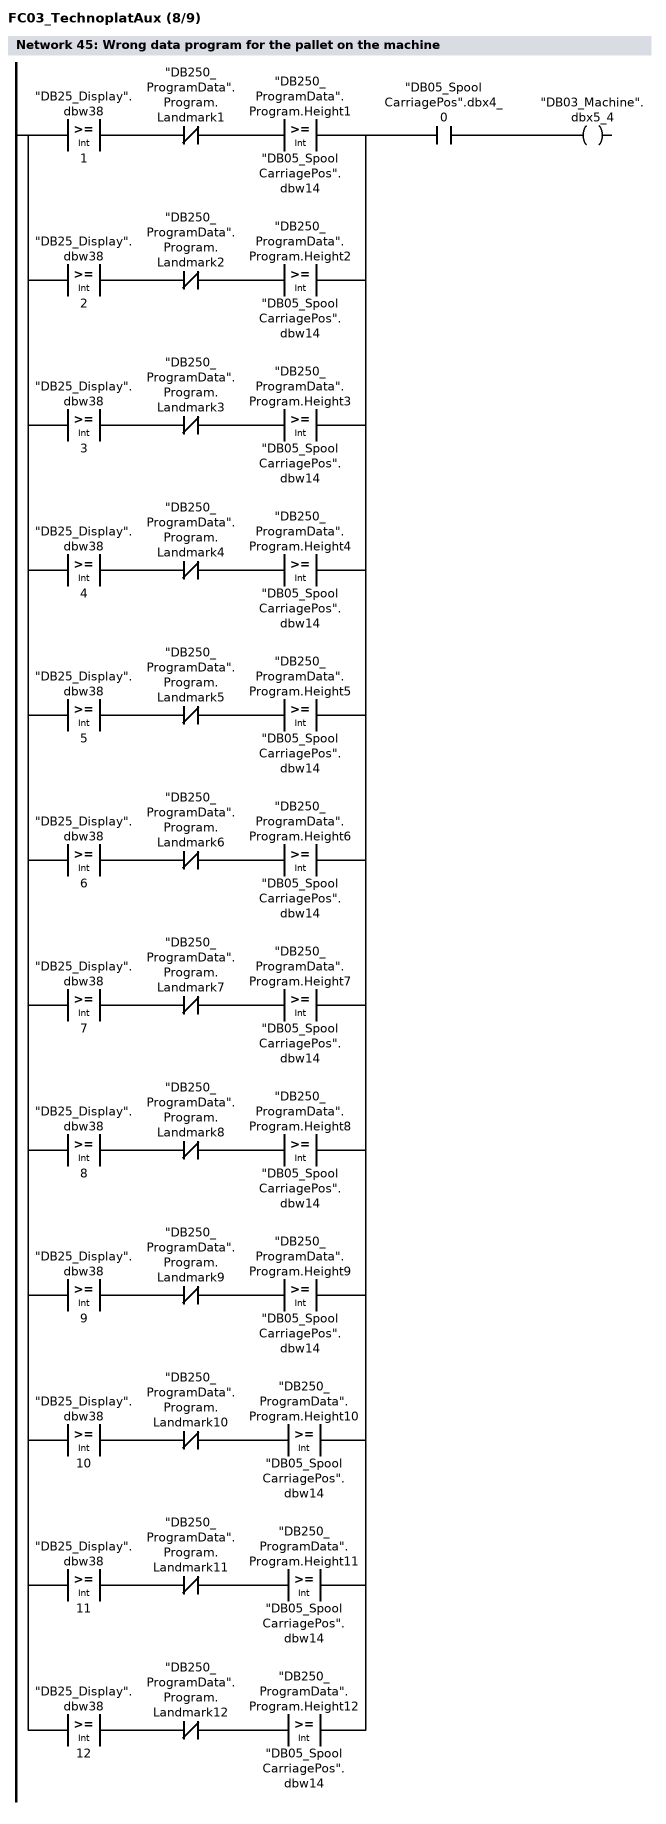
   RUNG wire#powerrail
      { S7_Templates := "SrcType := Int" } GE_Contact(in1 := "DB25_Display".dbw38, in2 := 1)
      I_Contact( "DB250_ProgramData".Program.Landmark1 )
      { S7_Templates := "SrcType := Int" } GE_Contact(in1 := "DB250_ProgramData".Program.Height1, in2 := "DB05_SpoolCarriagePos".dbw14)
      wire#w1
      Contact( "DB05_SpoolCarriagePos".dbx4_0 )
      Coil( "DB03_Machine".dbx5_4 )
   END_RUNG
   RUNG wire#powerrail
      { S7_Templates := "SrcType := Int" } GE_Contact(in1 := "DB25_Display".dbw38, in2 := 2)
      I_Contact( "DB250_ProgramData".Program.Landmark2 )
      { S7_Templates := "SrcType := Int" } GE_Contact(in1 := "DB250_ProgramData".Program.Height2, in2 := "DB05_SpoolCarriagePos".dbw14)
   END_RUNG wire#w1
   RUNG wire#powerrail
      { S7_Templates := "SrcType := Int" } GE_Contact(in1 := "DB25_Display".dbw38, in2 := 3)
      I_Contact( "DB250_ProgramData".Program.Landmark3 )
      { S7_Templates := "SrcType := Int" } GE_Contact(in1 := "DB250_ProgramData".Program.Height3, in2 := "DB05_SpoolCarriagePos".dbw14)
   END_RUNG wire#w1
   RUNG wire#powerrail
      { S7_Templates := "SrcType := Int" } GE_Contact(in1 := "DB25_Display".dbw38, in2 := 4)
      I_Contact( "DB250_ProgramData".Program.Landmark4 )
      { S7_Templates := "SrcType := Int" } GE_Contact(in1 := "DB250_ProgramData".Program.Height4, in2 := "DB05_SpoolCarriagePos".dbw14)
   END_RUNG wire#w1
   RUNG wire#powerrail
      { S7_Templates := "SrcType := Int" } GE_Contact(in1 := "DB25_Display".dbw38, in2 := 5)
      I_Contact( "DB250_ProgramData".Program.Landmark5 )
      { S7_Templates := "SrcType := Int" } GE_Contact(in1 := "DB250_ProgramData".Program.Height5, in2 := "DB05_SpoolCarriagePos".dbw14)
   END_RUNG wire#w1
   RUNG wire#powerrail
      { S7_Templates := "SrcType := Int" } GE_Contact(in1 := "DB25_Display".dbw38, in2 := 6)
      I_Contact( "DB250_ProgramData".Program.Landmark6 )
      { S7_Templates := "SrcType := Int" } GE_Contact(in1 := "DB250_ProgramData".Program.Height6, in2 := "DB05_SpoolCarriagePos".dbw14)
   END_RUNG wire#w1
   RUNG wire#powerrail
      { S7_Templates := "SrcType := Int" } GE_Contact(in1 := "DB25_Display".dbw38, in2 := 7)
      I_Contact( "DB250_ProgramData".Program.Landmark7 )
      { S7_Templates := "SrcType := Int" } GE_Contact(in1 := "DB250_ProgramData".Program.Height7, in2 := "DB05_SpoolCarriagePos".dbw14)
   END_RUNG wire#w1
   RUNG wire#powerrail
      { S7_Templates := "SrcType := Int" } GE_Contact(in1 := "DB25_Display".dbw38, in2 := 8)
      I_Contact( "DB250_ProgramData".Program.Landmark8 )
      { S7_Templates := "SrcType := Int" } GE_Contact(in1 := "DB250_ProgramData".Program.Height8, in2 := "DB05_SpoolCarriagePos".dbw14)
   END_RUNG wire#w1
   RUNG wire#powerrail
      { S7_Templates := "SrcType := Int" } GE_Contact(in1 := "DB25_Display".dbw38, in2 := 9)
      I_Contact( "DB250_ProgramData".Program.Landmark9 )
      { S7_Templates := "SrcType := Int" } GE_Contact(in1 := "DB250_ProgramData".Program.Height9, in2 := "DB05_SpoolCarriagePos".dbw14)
   END_RUNG wire#w1
   RUNG wire#powerrail
      { S7_Templates := "SrcType := Int" } GE_Contact(in1 := "DB25_Display".dbw38, in2 := 10)
      I_Contact( "DB250_ProgramData".Program.Landmark10 )
      { S7_Templates := "SrcType := Int" } GE_Contact(in1 := "DB250_ProgramData".Program.Height10, in2 := "DB05_SpoolCarriagePos".dbw14)
   END_RUNG wire#w1
   RUNG wire#powerrail
      { S7_Templates := "SrcType := Int" } GE_Contact(in1 := "DB25_Display".dbw38, in2 := 11)
      I_Contact( "DB250_ProgramData".Program.Landmark11 )
      { S7_Templates := "SrcType := Int" } GE_Contact(in1 := "DB250_ProgramData".Program.Height11, in2 := "DB05_SpoolCarriagePos".dbw14)
   END_RUNG wire#w1
   RUNG wire#powerrail
      { S7_Templates := "SrcType := Int" } GE_Contact(in1 := "DB25_Display".dbw38, in2 := 12)
      I_Contact( "DB250_ProgramData".Program.Landmark12 )
      { S7_Templates := "SrcType := Int" } GE_Contact(in1 := "DB250_ProgramData".Program.Height12, in2 := "DB05_SpoolCarriagePos".dbw14)
   END_RUNG wire#w1
   // the same network as SCL:
   "DB03_Machine".dbx5_4 := ((("DB25_Display".dbw38 >= 1) AND NOT "DB250_ProgramData".Program.Landmark1 AND ("DB250_ProgramData".Program.Height1 >= "DB05_SpoolCarriagePos".dbw14)) OR (("DB25_Display".dbw38 >= 2) AND NOT "DB250_ProgramData".Program.Landmark2 AND ("DB250_ProgramData".Program.Height2 >= "DB05_SpoolCarriagePos".dbw14)) OR (("DB25_Display".dbw38 >= 3) AND NOT "DB250_ProgramData".Program.Landmark3 AND ("DB250_ProgramData".Program.Height3 >= "DB05_SpoolCarriagePos".dbw14)) OR (("DB25_Display".dbw38 >= 4) AND NOT "DB250_ProgramData".Program.Landmark4 AND ("DB250_ProgramData".Program.Height4 >= "DB05_SpoolCarriagePos".dbw14)) OR (("DB25_Display".dbw38 >= 5) AND NOT "DB250_ProgramData".Program.Landmark5 AND ("DB250_ProgramData".Program.Height5 >= "DB05_SpoolCarriagePos".dbw14)) OR (("DB25_Display".dbw38 >= 6) AND NOT "DB250_ProgramData".Program.Landmark6 AND ("DB250_ProgramData".Program.Height6 >= "DB05_SpoolCarriagePos".dbw14)) OR (("DB25_Display".dbw38 >= 7) AND NOT "DB250_ProgramData".Program.Landmark7 AND ("DB250_ProgramData".Program.Height7 >= "DB05_SpoolCarriagePos".dbw14)) OR (("DB25_Display".dbw38 >= 8) AND NOT "DB250_ProgramData".Program.Landmark8 AND ("DB250_ProgramData".Program.Height8 >= "DB05_SpoolCarriagePos".dbw14)) OR (("DB25_Display".dbw38 >= 9) AND NOT "DB250_ProgramData".Program.Landmark9 AND ("DB250_ProgramData".Program.Height9 >= "DB05_SpoolCarriagePos".dbw14)) OR (("DB25_Display".dbw38 >= 10) AND NOT "DB250_ProgramData".Program.Landmark10 AND ("DB250_ProgramData".Program.Height10 >= "DB05_SpoolCarriagePos".dbw14)) OR (("DB25_Display".dbw38 >= 11) AND NOT "DB250_ProgramData".Program.Landmark11 AND ("DB250_ProgramData".Program.Height11 >= "DB05_SpoolCarriagePos".dbw14)) OR (("DB25_Display".dbw38 >= 12) AND NOT "DB250_ProgramData".Program.Landmark12 AND ("DB250_ProgramData".Program.Height12 >= "DB05_SpoolCarriagePos".dbw14))) AND "DB05_SpoolCarriagePos".dbx4_0;
END_REGION

REGION Network 46: Automatic mode for external conveyors
   // il transito tra 4 e 5 va sempre completato (in caso di richiesta E118 o porta non aperta /E119)
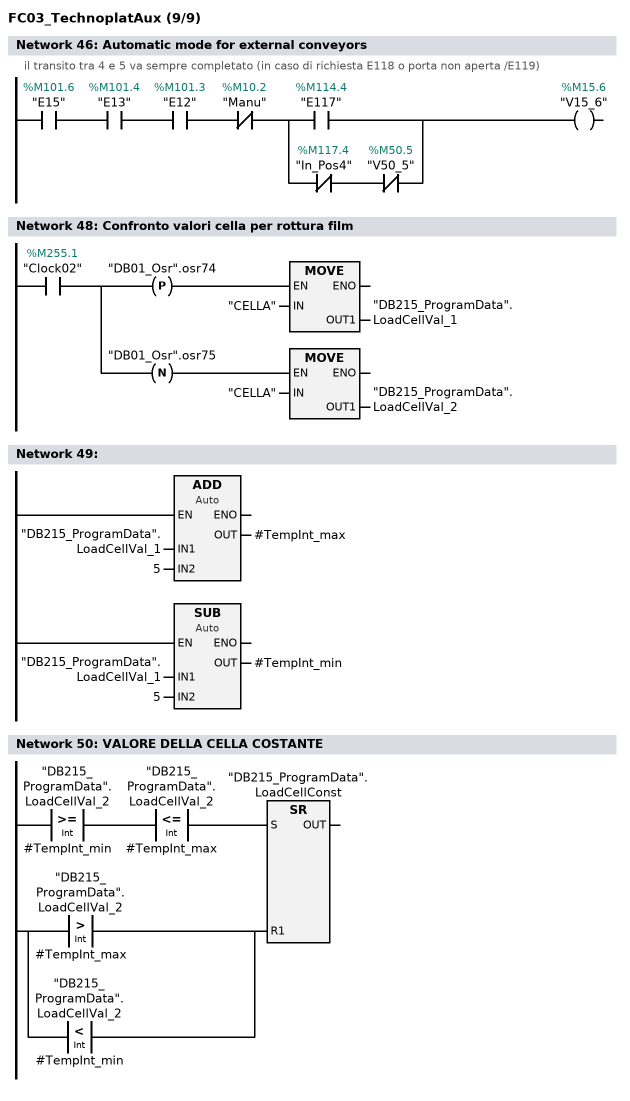
   RUNG wire#powerrail
      Contact( "E15" )
      Contact( "E13" )
      Contact( "E12" )
      I_Contact( "Manu" )
      wire#w1
      Contact( "E117" )
      wire#w2
      Coil( "V15_6" )
   END_RUNG
   RUNG wire#w1
      I_Contact( "In_Pos4" )
      I_Contact( "V50_5" )
   END_RUNG wire#w2
   // the same network as SCL:
   "V15_6" := "E15" AND "E13" AND "E12" AND NOT "Manu" AND ("E117" OR (NOT "In_Pos4" AND NOT "V50_5"));
END_REGION

REGION Network 47: ROTTURA FILM
END_REGION

REGION Network 48: Confronto valori cella per rottura film
   RUNG wire#powerrail
      Contact( "Clock02" )
      wire#w1
      P_Trig( "DB01_Osr".osr74 )
      Move(in := "CELLA", out1 => "DB215_ProgramData".LoadCellVal_1)
   END_RUNG
   RUNG wire#w1
      N_Trig( "DB01_Osr".osr75 )
      Move(in := "CELLA", out1 => "DB215_ProgramData".LoadCellVal_2)
   END_RUNG
   // the same network as SCL:
   #_w1 := "Clock02" AND NOT "DB01_Osr".osr74;   // rising edge
   "DB01_Osr".osr74 := "Clock02";
   IF #_w1 THEN "DB215_ProgramData".LoadCellVal_1 := "CELLA"; END_IF;
   #_w2 := NOT "Clock02" AND "DB01_Osr".osr75;   // falling edge
   "DB01_Osr".osr75 := "Clock02";
   IF #_w2 THEN "DB215_ProgramData".LoadCellVal_2 := "CELLA"; END_IF;
END_REGION

REGION Network 49
   RUNG wire#powerrail
      Add(in1 := "DB215_ProgramData".LoadCellVal_1, in2 := 5, out => #TempInt_max)
   END_RUNG
   RUNG wire#powerrail
      Sub(in1 := "DB215_ProgramData".LoadCellVal_1, in2 := 5, out => #TempInt_min)
   END_RUNG
   // the same network as SCL:
   #TempInt_max := "DB215_ProgramData".LoadCellVal_1 + 5;
   #TempInt_min := "DB215_ProgramData".LoadCellVal_1 - 5;
END_REGION

REGION Network 50: VALORE DELLA CELLA COSTANTE
   RUNG wire#powerrail
      { S7_Templates := "SrcType := Int" } GE_Contact(in1 := "DB215_ProgramData".LoadCellVal_2, in2 := #TempInt_min)
      { S7_Templates := "SrcType := Int" } LE_Contact(in1 := "DB215_ProgramData".LoadCellVal_2, in2 := #TempInt_max)
      S_SR(operand := "DB215_ProgramData".LoadCellConst, r1 := wire#w1)
   END_RUNG
   RUNG wire#powerrail
      { S7_Templates := "SrcType := Int" } GT_Contact(in1 := "DB215_ProgramData".LoadCellVal_2, in2 := #TempInt_max)
   END_RUNG wire#w1
   RUNG wire#powerrail
      { S7_Templates := "SrcType := Int" } LT_Contact(in1 := "DB215_ProgramData".LoadCellVal_2, in2 := #TempInt_min)
   END_RUNG wire#w1
   // the same network as SCL:
   IF ("DB215_ProgramData".LoadCellVal_2 >= #TempInt_min) AND ("DB215_ProgramData".LoadCellVal_2 <= #TempInt_max) THEN
       "DB215_ProgramData".LoadCellConst := TRUE;   // SR flip-flop
   END_IF;
   IF ("DB215_ProgramData".LoadCellVal_2 > #TempInt_max) OR ("DB215_ProgramData".LoadCellVal_2 < #TempInt_min) THEN
       "DB215_ProgramData".LoadCellConst := FALSE;
   END_IF;
END_REGION
END_FUNCTION

FUNCTION "FC100_BlockMoveIdexed" : Void
{ S7_Optimized_Access := 'FALSE' }
VERSION : 0.1
   VAR_INPUT 
      DBSource : Int;
      ByteSource : Int;
      DBDestination : Int;
      ByteDestination : Int;
      ByteNumber : Int;
   END_VAR


BEGIN
	POKE_BLK(area_src := 16#84,
	         dbNumber_src := #DBSource,
	         byteOffset_src := #ByteSource,
	         area_dest := 16#84,
	         dbNumber_dest := #DBDestination,
	         byteOffset_dest := #ByteDestination,
	         count := #ByteNumber);
	
	
	
END_FUNCTION

FUNCTION "FC33_Auxiliary_Memories" : Void
{ S7_Optimized_Access := 'TRUE' }
VERSION : 0.0
   VAR_TEMP 
      p_carr : DInt;
      TempDInt : DInt;
      TempDInt2 : DInt;
      TempDInt_MLC : DInt;
   END_VAR


BEGIN
	//Auxiliary memories pt.2
	//***********************
	(*
	//
	//CONDIZIONI PER EMERGENZA MACCHINA
	"EmergencyCondition" := (NOT "Main_EMG") OR
	                        (NOT "Thermic") OR  //EmergencyCode = 62
	                        "Alarm2" OR
	                        "Bumper";
	//
	*)
	//GESTIONE MALFUNZIONAMENTI INVERTER
	//FAULT (anomalia)
	IF ("Inverter_Data".U201.actual_fault = 16#0000) AND
	    ("Inverter_Data".U221.actual_fault = 16#0000) AND
	    ("Inverter_Data".U241.actual_fault = 16#0000) AND
	    ("Inverter_Data".U261.actual_fault = 16#0000) AND
	    ("Inverter_Data".U321.actual_fault = 16#0000) THEN
	    //    
	    "InverterFault" := 0;
	    "InverterFail" := 0;
	ELSE
	    "InverterFault" := 1;
	END_IF;
	//ALARM (avviso)
	IF ("Inverter_Data".U201.actual_alarm = 16#0000) AND
	    ("Inverter_Data".U221.actual_alarm = 16#0000) AND
	    ("Inverter_Data".U241.actual_alarm = 16#0000) AND
	    ("Inverter_Data".U261.actual_alarm = 16#0000) AND
	    ("Inverter_Data".U321.actual_alarm = 16#0000) THEN
	    //    
	    "InverterAlarm" := 0;
	ELSE    //copio il codice avviso (per poi visualizzarlo su HMI se persiste)
	    "Inverter_Alarms".U201_alarm := "Inverter_Data".U201.actual_alarm;
	    "Inverter_Alarms".U221_alarm := "Inverter_Data".U221.actual_alarm;
	    "Inverter_Alarms".U241_alarm := "Inverter_Data".U241.actual_alarm;
	    "Inverter_Alarms".U261_alarm := "Inverter_Data".U261.actual_alarm;
	    "Inverter_Alarms".U321_alarm := "Inverter_Data".U321.actual_alarm;
	    //    
	    "InverterAlarm" := 1;
	END_IF;
	//
	IF "Reset" THEN
	    "Inverter_Alarms".U201_alarm := 0;
	    "Inverter_Alarms".U221_alarm := 0;
	    "Inverter_Alarms".U241_alarm := 0;
	    "Inverter_Alarms".U261_alarm := 0;
	    "Inverter_Alarms".U321_alarm := 0;
	END_IF;
	//
	//Nel caso di "avvisi" attivo l'allarme solo se persistono per 5 secondi
	//
	IF ("InverterFault" OR "Timer".T200.Q) THEN
	    "InverterFail" := 1;
	    "DB23_AlarmProgram".dbx0_4 := 1;
	END_IF;
	//RESET (ACK)
	IF "Timer".T4.Q THEN
	    "U201_Ack" := 1;
	    "U221_Ack" := 1;
	    "U241_Ack" := 1;
	    "U261_Ack" := 1;
	    "U321_Ack" := 1;
	ELSE
	    "U201_Ack" := 0;
	    "U221_Ack" := 0;
	    "U241_Ack" := 0;
	    "U261_Ack" := 0;
	    "U321_Ack" := 0;
	END_IF;
	//
	//GESTIONE CELLA DI CARICO
	//************************
	(**)
	"CELLA" := "MB_REG1".A08R.REG_0; //(FC320_PID)
	//"CELLA" := 450; //(FC320_PID)
	//Reset cella
	IF "ResetLoadCell" THEN
	    "DB215_ProgramData".Offset_cella := "CELLA" + "DB215_ProgramData".ValOffsetCella;
	END_IF;
	//
	//APPOGGIO PER GRAFICO PID
	//*****
	//ROSA
	"DB100_Display".CELLA := ("CELLA" - 100) / 8;  //cella carico
	//ROSSO
	"DB100_Display".SETPOINT := ("DB320_PID".PID.setPointShow - 100) / 8;  //sp calcolato (cella)
	//VERDE
	"DB100_Display".PROP := (1 * DINT_TO_INT("DB320_PID".PID.proporzionale)) / 2;  //proporzionale
	//GIALLO
	"DB100_Display"."INT" := (1 * DINT_TO_INT("DB320_PID".PID.integrativo)) / 3;  //integrale
	//
	//AZZURRO
	"DB100_Display".FREQ_TIRO := (REAL_TO_INT("Inverter_Data".U241.setpoint)) / 30;  //integrale
	//AZZURRO
	"DB100_Display".FREQ_PRES := (REAL_TO_INT("Inverter_Data".U261.setpoint)) / 30;  //integrale
	//
	(*
	//
	//MOTORIZZAZIONI
	//Passi carrello + rotazione
	IF "DB230_Parameters".MotorType THEN
	    //SEW
	    "DB20_DisplaySysdata".dbd0 := 3730; 
	    "DB20_DisplaySysdata".dbd80 := 3180;
	ELSE //STD
	    "DB20_DisplaySysdata".dbd0 := 3330;
	    "DB20_DisplaySysdata".dbd80 := 7230; //enc.non integrato (P1)
	END_IF;
	//
	//Costanti per proporzioni velocità 
	"DB215_ProgramData".PropArmMax := 1770; //braccio@15rpm
	"DB215_ProgramData".PropCarrMax := 1933; //carrello@7.2m/min=120mm/s
	//
	//GESTIONE BRACCIO
	//****************
	//Zona sicurezza braccio (fuori ingombro)
	//
	IF "DB09_ArmPos".dbw34 > 3200 OR "DB09_ArmPos".dbw34 < 460 THEN
	    "SafetyPhase" := 1;
	ELSE
	    "SafetyPhase" := 0;
	END_IF;
	//
	//FASE DI TAGLIO
	//IF "DB09_ArmPos".dbw34 > 350 AND "DB09_ArmPos".dbw34 < 380 THEN
	IF ("DB09_ArmPos".dbw34 > ("DB230_Parameters".Cut_Phase - "DB20_DisplaySysdata".dbw84)) AND
	   ("DB09_ArmPos".dbw34 < ("DB230_Parameters".Cut_Phase + "DB20_DisplaySysdata".dbw84)) THEN
	    "CutPhase" := 1;
	ELSE
	    "CutPhase" := 0;
	END_IF;
	//
	//Velocità rotazione
	"DB215_ProgramData".RotSpeed := USINT_TO_INT("DB216_ActiveRecipe".Recipe.RotSpeed) * "DB215_ProgramData".PropArmMax / 15;
	//
	//Calcoli per decelerazione
	//Durata di un giro in ms in base alla velocità (60.000 msec / velocità in rpm)
	(*
	IF NOT "DB215_ProgramData".ActiveRecipeMLC THEN
	    "DB215_ProgramData".RoundTime := 60000 / USINT_TO_UINT("DB216_ActiveRecipe".Recipe.RotSpeed);
	ELSE
	    "DB215_ProgramData".RoundTime := 60000 / USINT_TO_UINT("DB216_ActiveRecipe".Recipe.MLC_L9.RotSpeed);
	END_IF;
	*)
	"DIAGNOSTICA".int_19 := INT_TO_UINT("DIAGNOSTICA".int_09);
	"DB215_ProgramData".RoundTime := 6000 / "DIAGNOSTICA".int_19; //decimi
	//Aumento il tempo in cui iniziare la decelerazione al diminuire della velocità (ci mette meno a fermarsi)
	//
	(*
	IF NOT "DB215_ProgramData".ActiveRecipeMLC THEN
	    #TempDInt := 125 - 5 * "DB216_ActiveRecipe".Recipe.RotSpeed; //(% di tempo giro) [(50:90) per (15:7)rpm]
	ELSE
	    #TempDInt := 125 - 5 * "DB216_ActiveRecipe".Recipe.MLC_L9.RotSpeed; //(% di tempo giro) [(50:90) per (15:7)rpm]
	END_IF;
	*)
	#TempDInt := 1250 - 5 * ("DIAGNOSTICA".int_19); //(% di tempo giro) [(50:90) per (15:7)rpm]
	#TempDInt2 := 60000 / "DIAGNOSTICA".int_19;//"DB215_ProgramData".RoundTime;    //T_giro
	"DB215_ProgramData".LastRoundTime := DINT_TO_UINT((#TempDInt * #TempDInt2) / 100);  //millisec
	//
	//GESTIONE CARRELLO
	//*****************
	//Direzione conteggio
	IF "FlagCarUp" THEN
	    "DB215_ProgramData".EncCarrDir := 1; //direzione conteggio UP
	ELSE
	    "DB215_ProgramData".EncCarrDir := -1; //direzione conteggio DOWN
	END_IF;
	//
	//Velocità salita/discesa
	#TempDInt := USINT_TO_DINT("DB216_ActiveRecipe".Recipe.CarSpeedUp) * "DB215_ProgramData".PropCarrMax / 72;
	"DB215_ProgramData".CarSpeedUp := DINT_TO_INT(#TempDInt);
	//
	#TempDInt := USINT_TO_DINT("DB216_ActiveRecipe".Recipe.CarSpeedDw) * "DB215_ProgramData".PropCarrMax / 72;
	"DB215_ProgramData".CarSpeedDw := DINT_TO_INT(#TempDInt);
	//
	//POSIZIONAMENTI CARRELLO
	//Passo [mm/1000p]
	#p_carr := "DB20_DisplaySysdata".dbd0;
	//
	//Altimetro
	#TempDInt := UINT_TO_DINT("DB216_ActiveRecipe".Recipe.Altimeter - 50) * 10000;
	"DB215_ProgramData".Altimeter_Pulses := DINT_TO_INT(#TempDInt / #p_carr);
	//
	//Ritardo fotocellula [ciclo STD; per MLC vedi FC33]
	//(se ho attivo il pressore considero lo spessore di circa 8 cm in meno del piatto)
	IF "DB216_ActiveRecipe".Recipe.PresserEnable THEN
	    IF "DB216_ActiveRecipe".Recipe.PhotDelay >= 8 THEN
	        #TempDInt := USINT_TO_DINT("DB216_ActiveRecipe".Recipe.PhotDelay - 8) * 10000;
	    ELSE
	        #TempDInt := USINT_TO_DINT("DB216_ActiveRecipe".Recipe.PhotDelay) * 10000;
	    END_IF;
	ELSE
	    #TempDInt := USINT_TO_DINT("DB216_ActiveRecipe".Recipe.PhotDelay) * 10000;
	END_IF;
	"DB215_ProgramData".PhotDelay_Pulses := DINT_TO_INT(#TempDInt / #p_carr);
	//
	//Giri rinforzo
	#TempDInt := USINT_TO_DINT("DB216_ActiveRecipe".Recipe.ReinforceHeight) * 10000;
	"DB215_ProgramData".Reinforce_Pulses := DINT_TO_INT(#TempDInt / #p_carr);
	//Discesa carrello per top
	#TempDInt := INT_TO_DINT("DB230_Parameters".TopCarrDescent) * 10000;
	"DB215_ProgramData".TopFall_Pulses := DINT_TO_INT(#TempDInt / #p_carr);
	//MLC
	//Forzamento a zero dell'ultimo strato (sempre in basso)
	"DB216_ActiveRecipe".Recipe.MLC_L9.Height := 0;
	//
	//Altezza strati (in base allo step del ciclo MLC) - Carica dati dello strato successivo
	IF "DB215_ProgramData".ActiveRecipeMLC THEN
	    CASE "DB200_Supervisor".State_Auto OF
	        15:
	            #TempDInt_MLC := UINT_TO_DINT("DB216_ActiveRecipe".Recipe.MLC_L1.Height) * 10000;
	            "DB215_ProgramData".MLC_HeightPulses := DINT_TO_INT(#TempDInt_MLC / #p_carr);
	//-----------------------------------------------------------------------------------------------            
	        212:
	            #TempDInt_MLC := UINT_TO_DINT("DB216_ActiveRecipe".Recipe.MLC_L2.Height) * 10000;
	            "DB215_ProgramData".MLC_HeightPulses := DINT_TO_INT(#TempDInt_MLC / #p_carr);
	//-----------------------------------------------------------------------------------------------            
	        220:
	            #TempDInt_MLC := UINT_TO_DINT("DB216_ActiveRecipe".Recipe.MLC_L2.Height) * 10000;
	            "DB215_ProgramData".MLC_HeightPulses := DINT_TO_INT(#TempDInt_MLC / #p_carr);
	        222:
	            #TempDInt_MLC := UINT_TO_DINT("DB216_ActiveRecipe".Recipe.MLC_L3.Height) * 10000;
	            "DB215_ProgramData".MLC_HeightPulses := DINT_TO_INT(#TempDInt_MLC / #p_carr);
	//-----------------------------------------------------------------------------------------------             
	        230:
	            #TempDInt_MLC := UINT_TO_DINT("DB216_ActiveRecipe".Recipe.MLC_L3.Height) * 10000;
	            "DB215_ProgramData".MLC_HeightPulses := DINT_TO_INT(#TempDInt_MLC / #p_carr);
	        232:
	            #TempDInt_MLC := UINT_TO_DINT("DB216_ActiveRecipe".Recipe.MLC_L4.Height) * 10000;
	            "DB215_ProgramData".MLC_HeightPulses := DINT_TO_INT(#TempDInt_MLC / #p_carr);
	//----------------------------------------------------------------------------------------------- 
	        240:
	            #TempDInt_MLC := UINT_TO_DINT("DB216_ActiveRecipe".Recipe.MLC_L4.Height) * 10000;
	            "DB215_ProgramData".MLC_HeightPulses := DINT_TO_INT(#TempDInt_MLC / #p_carr);
	        242:
	            #TempDInt_MLC := UINT_TO_DINT("DB216_ActiveRecipe".Recipe.MLC_L5.Height - 50) * 10000;
	            "DB215_ProgramData".MLC_HeightPulses := DINT_TO_INT(#TempDInt_MLC / #p_carr);
	//-----------------------------------------------------------------------------------------------     
	        255:
	            #TempDInt_MLC := UINT_TO_DINT("DB216_ActiveRecipe".Recipe.MLC_L6.Height) * 10000;
	            "DB215_ProgramData".MLC_HeightPulses := DINT_TO_INT(#TempDInt_MLC / #p_carr);
	//-----------------------------------------------------------------------------------------------    
	        260:
	            #TempDInt_MLC := UINT_TO_DINT("DB216_ActiveRecipe".Recipe.MLC_L6.Height) * 10000;
	            "DB215_ProgramData".MLC_HeightPulses := DINT_TO_INT(#TempDInt_MLC / #p_carr);
	        262:
	            #TempDInt_MLC := UINT_TO_DINT("DB216_ActiveRecipe".Recipe.MLC_L7.Height) * 10000;
	            "DB215_ProgramData".MLC_HeightPulses := DINT_TO_INT(#TempDInt_MLC / #p_carr);
	//-----------------------------------------------------------------------------------------------
	        270:
	            #TempDInt_MLC := UINT_TO_DINT("DB216_ActiveRecipe".Recipe.MLC_L7.Height) * 10000;
	            "DB215_ProgramData".MLC_HeightPulses := DINT_TO_INT(#TempDInt_MLC / #p_carr);
	        272:
	            #TempDInt_MLC := UINT_TO_DINT("DB216_ActiveRecipe".Recipe.MLC_L8.Height) * 10000;
	            "DB215_ProgramData".MLC_HeightPulses := DINT_TO_INT(#TempDInt_MLC / #p_carr);
	//-----------------------------------------------------------------------------------------------
	        280:
	            #TempDInt_MLC := UINT_TO_DINT("DB216_ActiveRecipe".Recipe.MLC_L8.Height) * 10000;
	            "DB215_ProgramData".MLC_HeightPulses := DINT_TO_INT(#TempDInt_MLC / #p_carr);
	        282:
	            #TempDInt_MLC := UINT_TO_DINT("DB216_ActiveRecipe".Recipe.MLC_L9.Height) * 10000;
	            "DB215_ProgramData".MLC_HeightPulses := DINT_TO_INT(#TempDInt_MLC / #p_carr);
	    END_CASE;
	   //
	END_IF;
	//
	//Lettura posizione carrello
	"DIAGNOSTICA".dint_01 := ("Enc_Carr" * #p_carr) / 10000;
	//
	//GESTIONE CICLO AUTOMATICO
	//*************************
	"ActiveCycle" := ("DB200_Supervisor".State_Auto >= 10); // <> 0);
	//
	//RESET CICLO (PULSANTE HMI) - SOLO MACCHINA
	"DB100_Display".CycleResetEnable := ("DB200_Supervisor".State_Stop = 170 AND
	(NOT "CutPhase" OR NOT "CarriageDown" //OR
	//(LPAS_enable AND NOT "CutArmBack")
	OR "ActiveCycle"));
	//
	//RESET CICLO MACCHINA
	IF "Reset" AND "Stop_state" THEN
	    "DB200_Supervisor".State_Auto := 0;
	END_IF;
	//
	//TIPO CICLO (con/senza top per Rototech3000)
	//
	IF "DB216_ActiveRecipe".Recipe.Cycle >= 3 THEN
	    "DB216_ActiveRecipe".Recipe.Cycle := 0;
	END_IF;
	//Con MLC non ha senso parlare di ciclo economico (solo waterproof)
	IF "DB215_ProgramData".ActiveRecipeMLC THEN
	    IF "DB216_ActiveRecipe".Recipe.Cycle >= 2 THEN
	        "DB216_ActiveRecipe".Recipe.Cycle := 0;
	    END_IF;
	END_IF;
	//No top
	IF "DB216_ActiveRecipe".Recipe.Cycle = 0 THEN
	    "DB03_Machine".TopBefore := 0;
	    "DB03_Machine".TopWaterP := 0;
	END_IF;
	//Top waterproof
	IF "DB216_ActiveRecipe".Recipe.Cycle = 1 THEN
	    "DB03_Machine".TopBefore := 0;
	    "DB03_Machine".TopWaterP := 1;
	END_IF;
	//Top dustproof (top before)
	IF "DB216_ActiveRecipe".Recipe.Cycle = 2 THEN
	    "DB03_Machine".TopBefore := 1;
	    "DB03_Machine".TopWaterP := 0;
	END_IF;
	//
	//RICETTE
	//Confronto ricette su HMI (modificabile) e PLC (salvata)
	IF (%DB216.DBD0 <> %DB229.DBD0 OR
	    %DB216.DBD4 <> %DB229.DBD4 OR
	    %DB216.DBD8 <> %DB229.DBD8 OR
	    %DB216.DBD12 <> %DB229.DBD12 OR
	    %DB216.DBD16 <> %DB229.DBD16 OR
	    %DB216.DBD20 <> %DB229.DBD20 OR
	    %DB216.DBD24 <> %DB229.DBD24 OR
	    %DB216.DBD28 <> %DB229.DBD28 OR
	    %DB216.DBD32 <> %DB229.DBD32 OR
	    %DB216.DBD36 <> %DB229.DBD36 OR
	    %DB216.DBD40 <> %DB229.DBD40 OR
	    %DB216.DBD44 <> %DB229.DBD44 OR
	    %DB216.DBD48 <> %DB229.DBD48 OR
	    %DB216.DBD52 <> %DB229.DBD52 OR
	    %DB216.DBD56 <> %DB229.DBD56 OR
	    %DB216.DBD60 <> %DB229.DBD60 OR
	    %DB216.DBD64 <> %DB229.DBD64 OR
	    %DB216.DBD68 <> %DB229.DBD68 OR
	    %DB216.DBD72 <> %DB229.DBD72 OR
	    %DB216.DBD76 <> %DB229.DBD76 OR
	    %DB216.DBD80 <> %DB229.DBD80 OR
	    %DB216.DBD84 <> %DB229.DBD84 OR
	    %DB216.DBD88 <> %DB229.DBD88 OR
	    %DB216.DBD92 <> %DB229.DBD92 OR
	    %DB216.DBD96 <> %DB229.DBD96 OR
	    %DB216.DBD100 <> %DB229.DBD100 OR
	    %DB216.DBD104 <> %DB229.DBD104 OR
	    %DB216.DBD108 <> %DB229.DBD108 OR
	    %DB216.DBD112 <> %DB229.DBD112 OR
	    %DB216.DBD116 <> %DB229.DBD116 OR
	    %DB216.DBD120 <> %DB229.DBD120 OR
	    %DB216.DBD124 <> %DB229.DBD124 OR
	    %DB216.DBD128 <> %DB229.DBD128 OR
	    %DB216.DBD132 <> %DB229.DBD132 OR
	    %DB216.DBD136 <> %DB229.DBD136 OR
	    %DB216.DBD140 <> %DB229.DBD140 OR
	    %DB216.DBD144 <> %DB229.DBD144 OR
	    %DB216.DBD148 <> %DB229.DBD148 OR
	    %DB216.DBD152 <> %DB229.DBD152 OR
	    %DB216.DBD156 <> %DB229.DBD156)
	THEN
	    "DB215_ProgramData".RecipeModified := 1;
	ELSE
	    "DB215_ProgramData".RecipeModified := 0;
	END_IF;
	//******************************************
	//LIMITI
	//Tiro
	IF ("DB216_ActiveRecipe".Recipe.StretchDwRounds < 0) THEN
	    "DB216_ActiveRecipe".Recipe.StretchDwRounds := 0;
	ELSIF ("DB216_ActiveRecipe".Recipe.StretchDwRounds > 100) THEN
	    "DB216_ActiveRecipe".Recipe.StretchDwRounds := 100;
	END_IF;
	//Forzamento del valore di tiro giri bassi su altri valori
	IF NOT "DB100_Display".TiroMultipleVal THEN
	    IF "DB216_ActiveRecipe".Recipe.StretchDwRounds <> "DB216_ActiveRecipe".Recipe.StretchUpward THEN
	        "DB216_ActiveRecipe".Recipe.StretchUpward := "DB216_ActiveRecipe".Recipe.StretchDwRounds;
	    END_IF;
	    IF "DB216_ActiveRecipe".Recipe.StretchDwRounds <> "DB216_ActiveRecipe".Recipe.StretchUpRounds THEN
	        "DB216_ActiveRecipe".Recipe.StretchUpRounds := "DB216_ActiveRecipe".Recipe.StretchDwRounds;
	    END_IF;
	    IF "DB216_ActiveRecipe".Recipe.StretchDwRounds <> "DB216_ActiveRecipe".Recipe.StretchDownward THEN
	        "DB216_ActiveRecipe".Recipe.StretchDownward := "DB216_ActiveRecipe".Recipe.StretchDwRounds;
	    END_IF;
	END_IF;
	//Prestiro
	IF ("DB216_ActiveRecipe".Recipe.Prestretch < 150) THEN
	    "DB216_ActiveRecipe".Recipe.Prestretch := 150;
	ELSIF ("DB216_ActiveRecipe".Recipe.Prestretch > 400) THEN
	    "DB216_ActiveRecipe".Recipe.Prestretch := 400;
	END_IF;
	// Velocità braccio
	IF ("DB216_ActiveRecipe".Recipe.RotSpeed < 7) THEN
	    "DB216_ActiveRecipe".Recipe.RotSpeed := 7;
	ELSIF ("DB216_ActiveRecipe".Recipe.RotSpeed > 15) THEN
	    "DB216_ActiveRecipe".Recipe.RotSpeed := 15;
	END_IF;
	// Velocità carrello
	IF ("DB216_ActiveRecipe".Recipe.CarSpeedUp < 25) THEN
	    "DB216_ActiveRecipe".Recipe.CarSpeedUp := 25;
	ELSIF ("DB216_ActiveRecipe".Recipe.CarSpeedUp > 72) THEN
	    "DB216_ActiveRecipe".Recipe.CarSpeedUp := 72;
	END_IF;
	IF ("DB216_ActiveRecipe".Recipe.CarSpeedDw < 25) THEN
	    "DB216_ActiveRecipe".Recipe.CarSpeedDw := 25;
	ELSIF ("DB216_ActiveRecipe".Recipe.CarSpeedDw > 72) THEN
	    "DB216_ActiveRecipe".Recipe.CarSpeedDw := 72;
	END_IF;
	//******************************************
	*)
END_FUNCTION

FUNCTION "FC08_SpoolCarriagePos" : Void   // FC8, LAD
TITLE = Spool carriages Helix40/2 positioning
{ S7_Optimized_Access := 'FALSE' }
AUTHOR : Robopac
VERSION : 0.0
// stored: AutoNumber false, IsIECCheckEnabled false, SetENOAutomatically false, UDAEnableTagReadback false
   VAR_TEMP
      Isteresi : Int;
      TempInt : Int;
      Encoder : Int;
      TempDint1 : DInt;
      TempWord : Word;
      TempDint2 : DInt;
   END_VAR
   VAR_TEMP   // added for the SCL form of the ladder/FBD networks
      _w1 : Bool;
      _w2 : Bool;
   END_VAR
BEGIN

REGION Network 1: Reset spool carriage positioning counter (pulse)
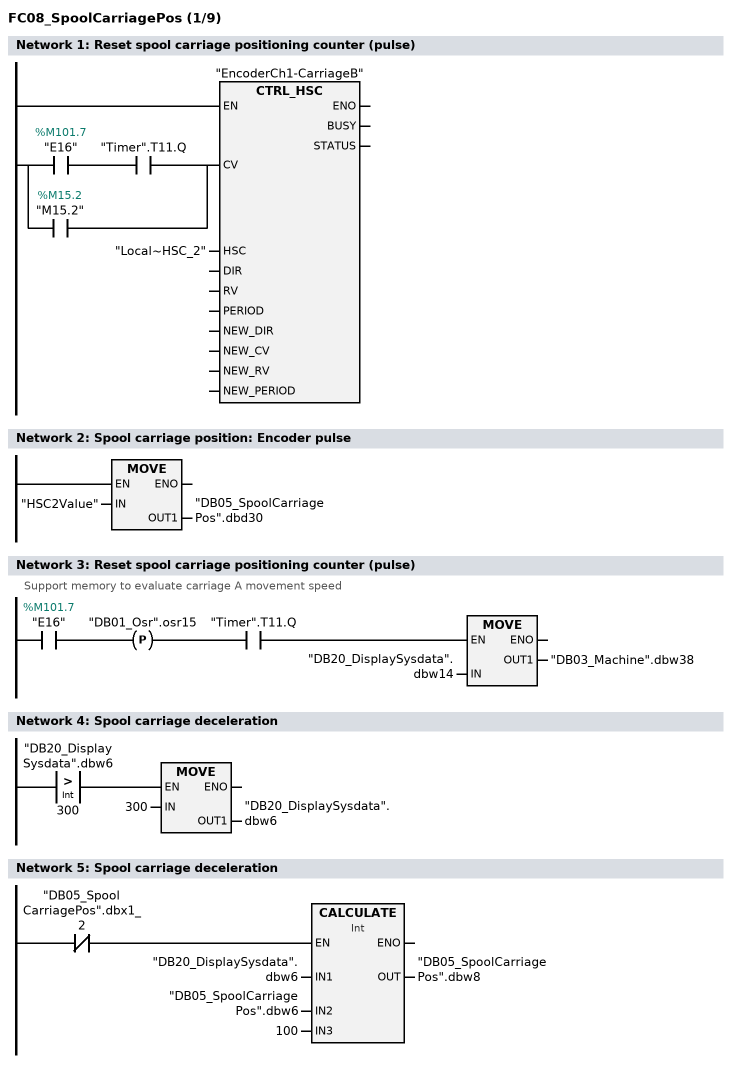
   RUNG wire#powerrail
      "EncoderCh1-CarriageB".CTRL_HSC(CV := wire#w1, HSC := "Local~HSC_2", DIR :=, RV :=, PERIOD :=, NEW_DIR :=, NEW_CV :=, NEW_RV :=, NEW_PERIOD :=, BUSY =>, STATUS =>)
   END_RUNG
   RUNG wire#powerrail
      Contact( "E16" )
      Contact( "Timer".T11.Q )
   END_RUNG wire#w1
   RUNG wire#powerrail
      Contact( "M15.2" )
   END_RUNG wire#w1
   // the same network as SCL:
   "EncoderCh1-CarriageB"(CV := ("E16" AND "Timer".T11.Q) OR "M15.2", HSC := "Local~HSC_2");   // CTRL_HSC
END_REGION

REGION Network 2: Spool carriage position: Encoder pulse
   RUNG wire#powerrail
      { S7_GenerateENO := "TRUE" } Move(in := "HSC2Value", out1 => "DB05_SpoolCarriagePos".dbd30)
   END_RUNG
   // the same network as SCL:
   "DB05_SpoolCarriagePos".dbd30 := "HSC2Value";
END_REGION

REGION Network 3: Reset spool carriage positioning counter (pulse)
   // Support memory to evaluate carriage A movement speed
   RUNG wire#powerrail
      Contact( "E16" )
      P_Trig( "DB01_Osr".osr15 )
      Contact( "Timer".T11.Q )
      { S7_GenerateENO := "TRUE" } Move(in := "DB20_DisplaySysdata".dbw14, out1 => "DB03_Machine".dbw38)
   END_RUNG
   // the same network as SCL:
   #_w1 := "E16" AND NOT "DB01_Osr".osr15;   // rising edge
   "DB01_Osr".osr15 := "E16";
   IF #_w1 AND "Timer".T11.Q THEN "DB03_Machine".dbw38 := "DB20_DisplaySysdata".dbw14; END_IF;
END_REGION

REGION Network 4: Spool carriage deceleration
   RUNG wire#powerrail
      { S7_Templates := "SrcType := Int" } GT_Contact(in1 := "DB20_DisplaySysdata".dbw6, in2 := 300)
      { S7_GenerateENO := "TRUE" } Move(in := 300, out1 => "DB20_DisplaySysdata".dbw6)
   END_RUNG
   // the same network as SCL:
   IF "DB20_DisplaySysdata".dbw6 > 300 THEN "DB20_DisplaySysdata".dbw6 := 300; END_IF;
END_REGION

REGION Network 5: Spool carriage deceleration
   RUNG wire#powerrail
      I_Contact( "DB05_SpoolCarriagePos".dbx1_2 )
      { S7_Templates := "SrcType := Int"; S7_GenerateENO := "TRUE"; S7_Expression := "In1 * In2 / In3" } Calculate(in1 := "DB20_DisplaySysdata".dbw6, in2 := "DB05_SpoolCarriagePos".dbw6, in3 := 100, out => "DB05_SpoolCarriagePos".dbw8)
   END_RUNG
   // the same network as SCL:
   IF NOT "DB05_SpoolCarriagePos".dbx1_2 THEN
       "DB05_SpoolCarriagePos".dbw8 := "DB20_DisplaySysdata".dbw6 * "DB05_SpoolCarriagePos".dbw6 / 100;
   END_IF;
END_REGION

REGION Network 6: Spool carriage position and deceleration
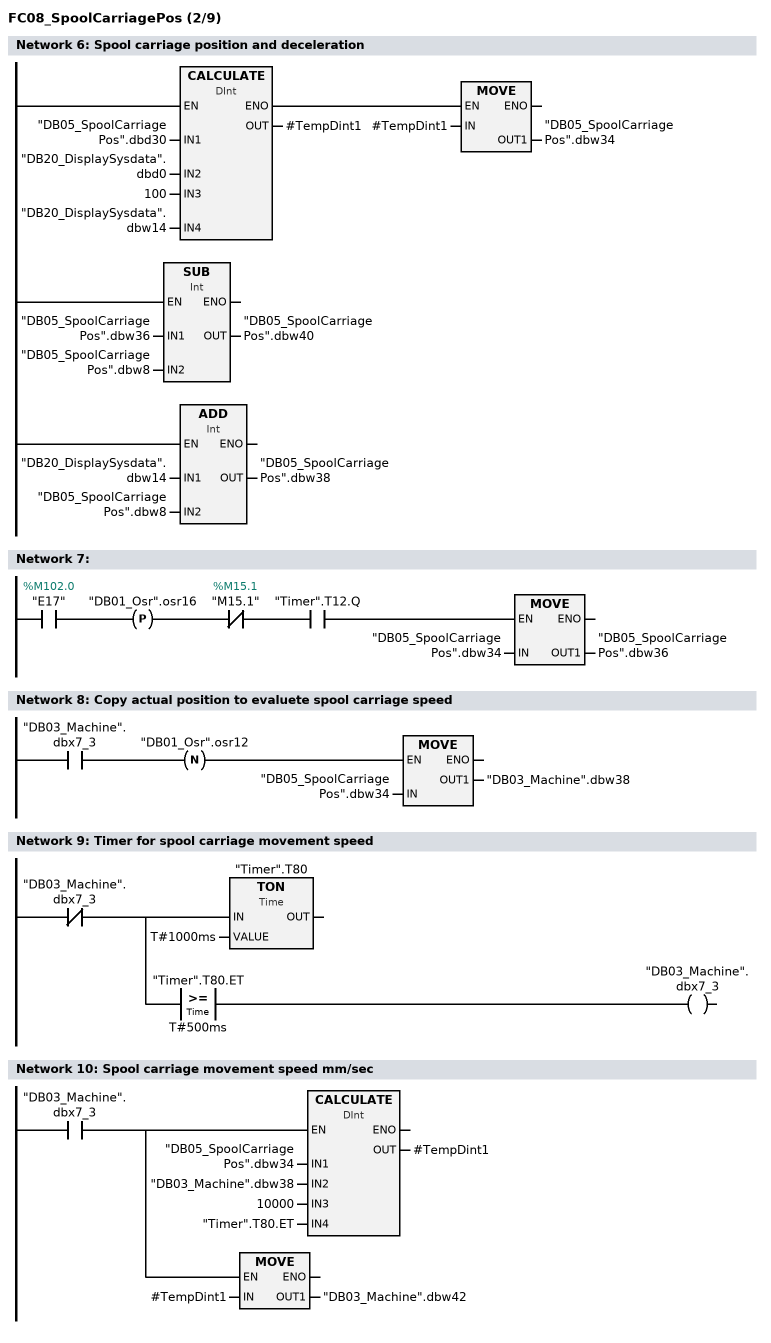
   RUNG wire#powerrail
      { S7_Templates := "SrcType := DInt"; S7_GenerateENO := "TRUE"; S7_Expression := "((In1*In2)/In3)+In4" } Calculate(in1 := "DB05_SpoolCarriagePos".dbd30, in2 := "DB20_DisplaySysdata".dbd0, in3 := 100, in4 := "DB20_DisplaySysdata".dbw14, out => #TempDint1)
      { S7_GenerateENO := "TRUE" } Move(in := #TempDint1, out1 => "DB05_SpoolCarriagePos".dbw34)
   END_RUNG
   RUNG wire#powerrail
      { S7_Templates := "SrcType := Int"; S7_GenerateENO := "TRUE" } Sub(in1 := "DB05_SpoolCarriagePos".dbw36, in2 := "DB05_SpoolCarriagePos".dbw8, out => "DB05_SpoolCarriagePos".dbw40)
   END_RUNG
   RUNG wire#powerrail
      { S7_Templates := "SrcType := Int"; S7_GenerateENO := "TRUE" } Add(in1 := "DB20_DisplaySysdata".dbw14, in2 := "DB05_SpoolCarriagePos".dbw8, out => "DB05_SpoolCarriagePos".dbw38)
   END_RUNG
   // the same network as SCL:
   // ENO of a box is taken as its EN; it also drops when the box reports an error
   #TempDint1 := (("DB05_SpoolCarriagePos".dbd30*"DB20_DisplaySysdata".dbd0)/100)+"DB20_DisplaySysdata".dbw14;
   "DB05_SpoolCarriagePos".dbw34 := #TempDint1;
   "DB05_SpoolCarriagePos".dbw40 := "DB05_SpoolCarriagePos".dbw36 - "DB05_SpoolCarriagePos".dbw8;
   "DB05_SpoolCarriagePos".dbw38 := "DB20_DisplaySysdata".dbw14 + "DB05_SpoolCarriagePos".dbw8;
END_REGION

REGION Network 7
   RUNG wire#powerrail
      Contact( "E17" )
      P_Trig( "DB01_Osr".osr16 )
      I_Contact( "M15.1" )
      Contact( "Timer".T12.Q )
      { S7_GenerateENO := "TRUE" } Move(in := "DB05_SpoolCarriagePos".dbw34, out1 => "DB05_SpoolCarriagePos".dbw36)
   END_RUNG
   // the same network as SCL:
   #_w1 := "E17" AND NOT "DB01_Osr".osr16;   // rising edge
   "DB01_Osr".osr16 := "E17";
   IF #_w1 AND NOT "M15.1" AND "Timer".T12.Q THEN
       "DB05_SpoolCarriagePos".dbw36 := "DB05_SpoolCarriagePos".dbw34;
   END_IF;
END_REGION

REGION Network 8: Copy actual position to evaluete spool carriage speed
   RUNG wire#powerrail
      Contact( "DB03_Machine".dbx7_3 )
      N_Trig( "DB01_Osr".osr12 )
      { S7_GenerateENO := "TRUE" } Move(in := "DB05_SpoolCarriagePos".dbw34, out1 => "DB03_Machine".dbw38)
   END_RUNG
   // the same network as SCL:
   #_w1 := NOT "DB03_Machine".dbx7_3 AND "DB01_Osr".osr12;   // falling edge
   "DB01_Osr".osr12 := "DB03_Machine".dbx7_3;
   IF #_w1 THEN "DB03_Machine".dbw38 := "DB05_SpoolCarriagePos".dbw34; END_IF;
END_REGION

REGION Network 9: Timer for spool carriage movement speed
   #_w1 := NOT "DB03_Machine".dbx7_3;
   "Timer".T80.TON(IN := #_w1, PT := T#1000ms);   // TON coil
   "DB03_Machine".dbx7_3 := #_w1 AND ("Timer".T80.ET >= T#500ms);
END_REGION

REGION Network 10: Spool carriage movement speed mm/sec
   RUNG wire#powerrail
      Contact( "DB03_Machine".dbx7_3 )
      wire#w1
      { S7_Templates := "SrcType := DInt"; S7_GenerateENO := "TRUE"; S7_Expression := "(In1-In2)*In3/In4" } Calculate(in1 := "DB05_SpoolCarriagePos".dbw34, in2 := "DB03_Machine".dbw38, in3 := 10000, in4 := "Timer".T80.ET, out => #TempDint1)
   END_RUNG
   RUNG wire#w1
      { S7_GenerateENO := "TRUE" } Move(in := #TempDint1, out1 => "DB03_Machine".dbw42)
   END_RUNG
   // the same network as SCL:
   IF "DB03_Machine".dbx7_3 THEN
       #TempDint1 := ("DB05_SpoolCarriagePos".dbw34-"DB03_Machine".dbw38)*10000/"Timer".T80.ET;
       "DB03_Machine".dbw42 := #TempDint1;
   END_IF;
END_REGION

REGION Network 11: Spool carriage movement speed mm/sec recorded
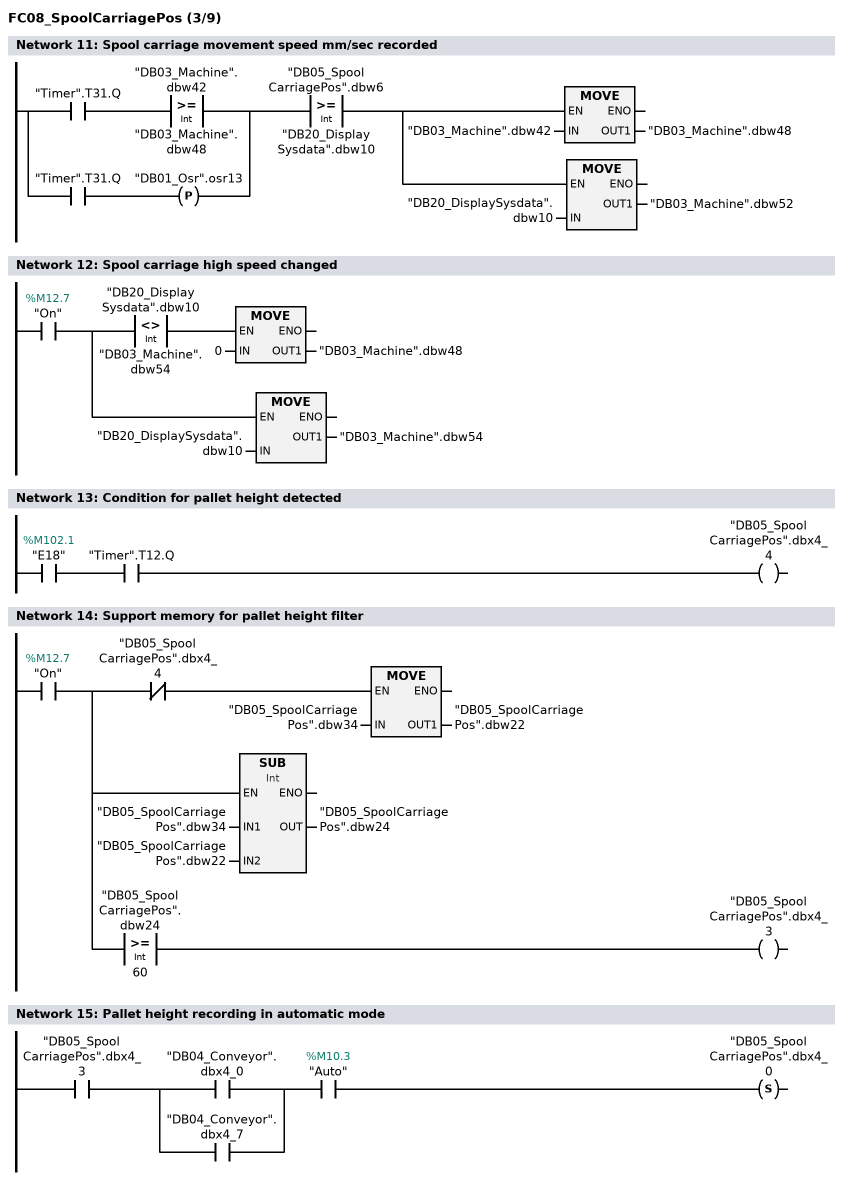
   RUNG wire#powerrail
      Contact( "Timer".T31.Q )
      { S7_Templates := "SrcType := Int" } GE_Contact(in1 := "DB03_Machine".dbw42, in2 := "DB03_Machine".dbw48)
      wire#w1
      { S7_Templates := "SrcType := Int" } GE_Contact(in1 := "DB05_SpoolCarriagePos".dbw6, in2 := "DB20_DisplaySysdata".dbw10)
      wire#w2
      { S7_GenerateENO := "TRUE" } Move(in := "DB03_Machine".dbw42, out1 => "DB03_Machine".dbw48)
   END_RUNG
   RUNG wire#powerrail
      Contact( "Timer".T31.Q )
      P_Trig( "DB01_Osr".osr13 )
   END_RUNG wire#w1
   RUNG wire#w2
      { S7_GenerateENO := "TRUE" } Move(in := "DB20_DisplaySysdata".dbw10, out1 => "DB03_Machine".dbw52)
   END_RUNG
   // the same network as SCL:
   #_w1 := "Timer".T31.Q AND NOT "DB01_Osr".osr13;   // rising edge
   "DB01_Osr".osr13 := "Timer".T31.Q;
   #_w2 := (("Timer".T31.Q AND ("DB03_Machine".dbw42 >= "DB03_Machine".dbw48)) OR #_w1) AND ("DB05_SpoolCarriagePos".dbw6 >= "DB20_DisplaySysdata".dbw10);
   IF #_w2 THEN
       "DB03_Machine".dbw48 := "DB03_Machine".dbw42;
       "DB03_Machine".dbw52 := "DB20_DisplaySysdata".dbw10;
   END_IF;
END_REGION

REGION Network 12: Spool carriage high speed changed
   RUNG wire#powerrail
      Contact( "On" )
      wire#w1
      { S7_Templates := "SrcType := Int" } NE_Contact(in1 := "DB20_DisplaySysdata".dbw10, in2 := "DB03_Machine".dbw54)
      { S7_GenerateENO := "TRUE" } Move(in := 0, out1 => "DB03_Machine".dbw48)
   END_RUNG
   RUNG wire#w1
      { S7_GenerateENO := "TRUE" } Move(in := "DB20_DisplaySysdata".dbw10, out1 => "DB03_Machine".dbw54)
   END_RUNG
   // the same network as SCL:
   IF "On" AND ("DB20_DisplaySysdata".dbw10 <> "DB03_Machine".dbw54) THEN "DB03_Machine".dbw48 := 0; END_IF;
   IF "On" THEN "DB03_Machine".dbw54 := "DB20_DisplaySysdata".dbw10; END_IF;
END_REGION

REGION Network 13: Condition for pallet height detected
   RUNG wire#powerrail
      Contact( "E18" )
      Contact( "Timer".T12.Q )
      Coil( "DB05_SpoolCarriagePos".dbx4_4 )
   END_RUNG
   // the same network as SCL:
   "DB05_SpoolCarriagePos".dbx4_4 := "E18" AND "Timer".T12.Q;
END_REGION

REGION Network 14: Support memory for pallet height filter
   RUNG wire#powerrail
      Contact( "On" )
      wire#w1
      I_Contact( "DB05_SpoolCarriagePos".dbx4_4 )
      { S7_GenerateENO := "TRUE" } Move(in := "DB05_SpoolCarriagePos".dbw34, out1 => "DB05_SpoolCarriagePos".dbw22)
   END_RUNG
   RUNG wire#w1
      { S7_Templates := "SrcType := Int"; S7_GenerateENO := "TRUE" } Sub(in1 := "DB05_SpoolCarriagePos".dbw34, in2 := "DB05_SpoolCarriagePos".dbw22, out => "DB05_SpoolCarriagePos".dbw24)
   END_RUNG
   RUNG wire#w1
      { S7_Templates := "SrcType := Int" } GE_Contact(in1 := "DB05_SpoolCarriagePos".dbw24, in2 := 60)
      Coil( "DB05_SpoolCarriagePos".dbx4_3 )
   END_RUNG
   // the same network as SCL:
   IF "On" AND NOT "DB05_SpoolCarriagePos".dbx4_4 THEN
       "DB05_SpoolCarriagePos".dbw22 := "DB05_SpoolCarriagePos".dbw34;
   END_IF;
   IF "On" THEN
       "DB05_SpoolCarriagePos".dbw24 := "DB05_SpoolCarriagePos".dbw34 - "DB05_SpoolCarriagePos".dbw22;
   END_IF;
   "DB05_SpoolCarriagePos".dbx4_3 := "On" AND ("DB05_SpoolCarriagePos".dbw24 >= 60);
END_REGION

REGION Network 15: Pallet height recording in automatic mode
   RUNG wire#powerrail
      Contact( "DB05_SpoolCarriagePos".dbx4_3 )
      wire#w1
      Contact( "DB04_Conveyor".dbx4_0 )
      wire#w2
      Contact( "Auto" )
      S_Coil( "DB05_SpoolCarriagePos".dbx4_0 )
   END_RUNG
   RUNG wire#w1
      Contact( "DB04_Conveyor".dbx4_7 )
   END_RUNG wire#w2
   // the same network as SCL:
   IF "DB05_SpoolCarriagePos".dbx4_3 AND ("DB04_Conveyor".dbx4_0 OR "DB04_Conveyor".dbx4_7) AND "Auto" THEN
       "DB05_SpoolCarriagePos".dbx4_0 := TRUE;
   END_IF;
END_REGION

REGION Network 16: Recording pallet height for wrapping position
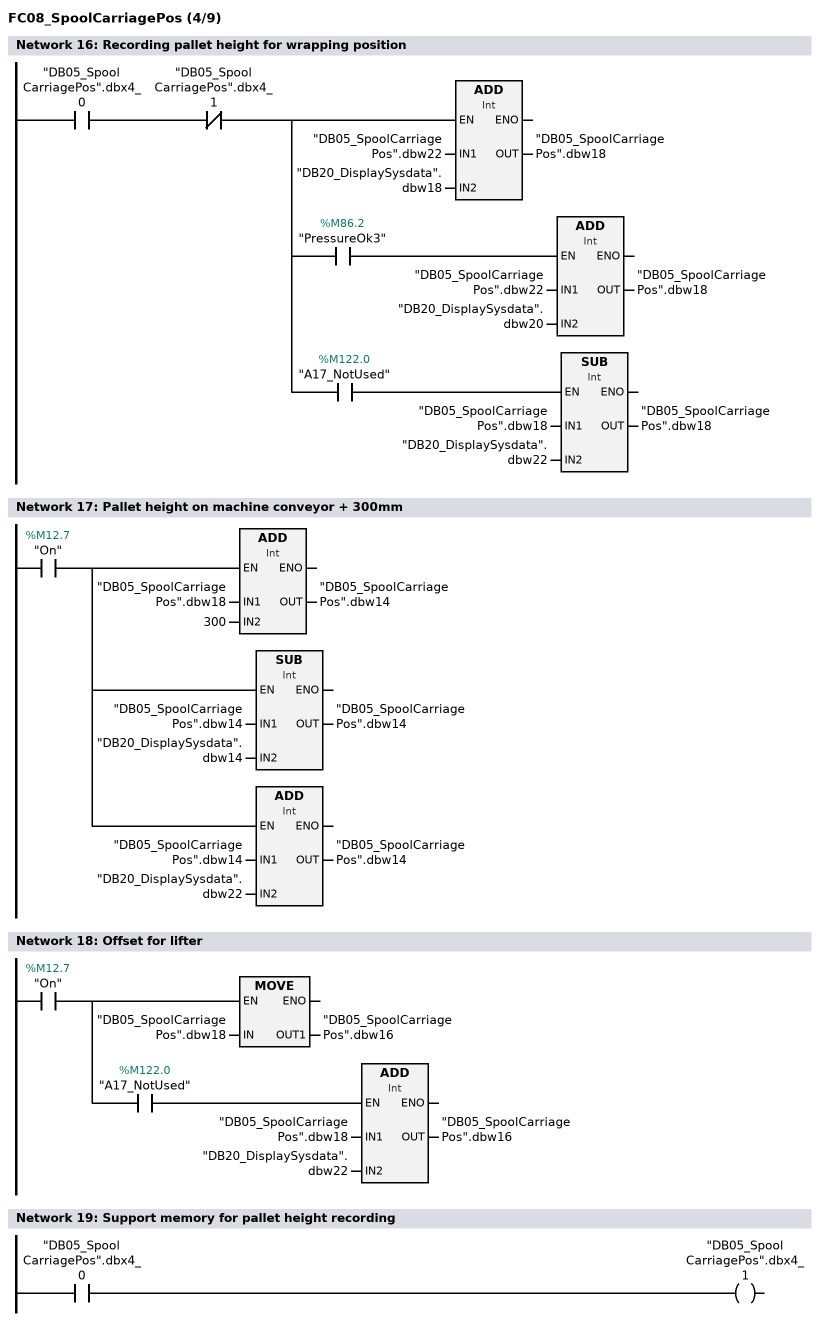
   RUNG wire#powerrail
      Contact( "DB05_SpoolCarriagePos".dbx4_0 )
      I_Contact( "DB05_SpoolCarriagePos".dbx4_1 )
      wire#w1
      { S7_Templates := "SrcType := Int"; S7_GenerateENO := "TRUE" } Add(in1 := "DB05_SpoolCarriagePos".dbw22, in2 := "DB20_DisplaySysdata".dbw18, out => "DB05_SpoolCarriagePos".dbw18)
   END_RUNG
   RUNG wire#w1
      Contact( "PressureOk3" )
      { S7_Templates := "SrcType := Int"; S7_GenerateENO := "TRUE" } Add(in1 := "DB05_SpoolCarriagePos".dbw22, in2 := "DB20_DisplaySysdata".dbw20, out => "DB05_SpoolCarriagePos".dbw18)
   END_RUNG
   RUNG wire#w1
      Contact( "A17_NotUsed" )
      { S7_Templates := "SrcType := Int"; S7_GenerateENO := "TRUE" } Sub(in1 := "DB05_SpoolCarriagePos".dbw18, in2 := "DB20_DisplaySysdata".dbw22, out => "DB05_SpoolCarriagePos".dbw18)
   END_RUNG
   // the same network as SCL:
   #_w1 := "DB05_SpoolCarriagePos".dbx4_0 AND NOT "DB05_SpoolCarriagePos".dbx4_1;
   IF #_w1 THEN
       "DB05_SpoolCarriagePos".dbw18 := "DB05_SpoolCarriagePos".dbw22 + "DB20_DisplaySysdata".dbw18;
   END_IF;
   IF #_w1 AND "PressureOk3" THEN
       "DB05_SpoolCarriagePos".dbw18 := "DB05_SpoolCarriagePos".dbw22 + "DB20_DisplaySysdata".dbw20;
   END_IF;
   IF #_w1 AND "A17_NotUsed" THEN
       "DB05_SpoolCarriagePos".dbw18 := "DB05_SpoolCarriagePos".dbw18 - "DB20_DisplaySysdata".dbw22;
   END_IF;
END_REGION

REGION Network 17: Pallet height on machine conveyor + 300mm
   RUNG wire#powerrail
      Contact( "On" )
      wire#w1
      { S7_Templates := "SrcType := Int"; S7_GenerateENO := "TRUE" } Add(in1 := "DB05_SpoolCarriagePos".dbw18, in2 := 300, out => "DB05_SpoolCarriagePos".dbw14)
   END_RUNG
   RUNG wire#w1
      { S7_Templates := "SrcType := Int"; S7_GenerateENO := "TRUE" } Sub(in1 := "DB05_SpoolCarriagePos".dbw14, in2 := "DB20_DisplaySysdata".dbw14, out => "DB05_SpoolCarriagePos".dbw14)
   END_RUNG
   RUNG wire#w1
      { S7_Templates := "SrcType := Int"; S7_GenerateENO := "TRUE" } Add(in1 := "DB05_SpoolCarriagePos".dbw14, in2 := "DB20_DisplaySysdata".dbw22, out => "DB05_SpoolCarriagePos".dbw14)
   END_RUNG
   // the same network as SCL:
   IF "On" THEN
       "DB05_SpoolCarriagePos".dbw14 := "DB05_SpoolCarriagePos".dbw18 + 300;
       "DB05_SpoolCarriagePos".dbw14 := "DB05_SpoolCarriagePos".dbw14 - "DB20_DisplaySysdata".dbw14;
       "DB05_SpoolCarriagePos".dbw14 := "DB05_SpoolCarriagePos".dbw14 + "DB20_DisplaySysdata".dbw22;
   END_IF;
END_REGION

REGION Network 18: Offset for lifter
   RUNG wire#powerrail
      Contact( "On" )
      wire#w1
      { S7_GenerateENO := "TRUE" } Move(in := "DB05_SpoolCarriagePos".dbw18, out1 => "DB05_SpoolCarriagePos".dbw16)
   END_RUNG
   RUNG wire#w1
      Contact( "A17_NotUsed" )
      { S7_Templates := "SrcType := Int"; S7_GenerateENO := "TRUE" } Add(in1 := "DB05_SpoolCarriagePos".dbw18, in2 := "DB20_DisplaySysdata".dbw22, out => "DB05_SpoolCarriagePos".dbw16)
   END_RUNG
   // the same network as SCL:
   IF "On" THEN "DB05_SpoolCarriagePos".dbw16 := "DB05_SpoolCarriagePos".dbw18; END_IF;
   IF "On" AND "A17_NotUsed" THEN
       "DB05_SpoolCarriagePos".dbw16 := "DB05_SpoolCarriagePos".dbw18 + "DB20_DisplaySysdata".dbw22;
   END_IF;
END_REGION

REGION Network 19: Support memory for pallet height recording
   RUNG wire#powerrail
      Contact( "DB05_SpoolCarriagePos".dbx4_0 )
      Coil( "DB05_SpoolCarriagePos".dbx4_1 )
   END_RUNG
   // the same network as SCL:
   "DB05_SpoolCarriagePos".dbx4_1 := "DB05_SpoolCarriagePos".dbx4_0;
END_REGION

REGION Network 20: Pallet height recording in automatic mode
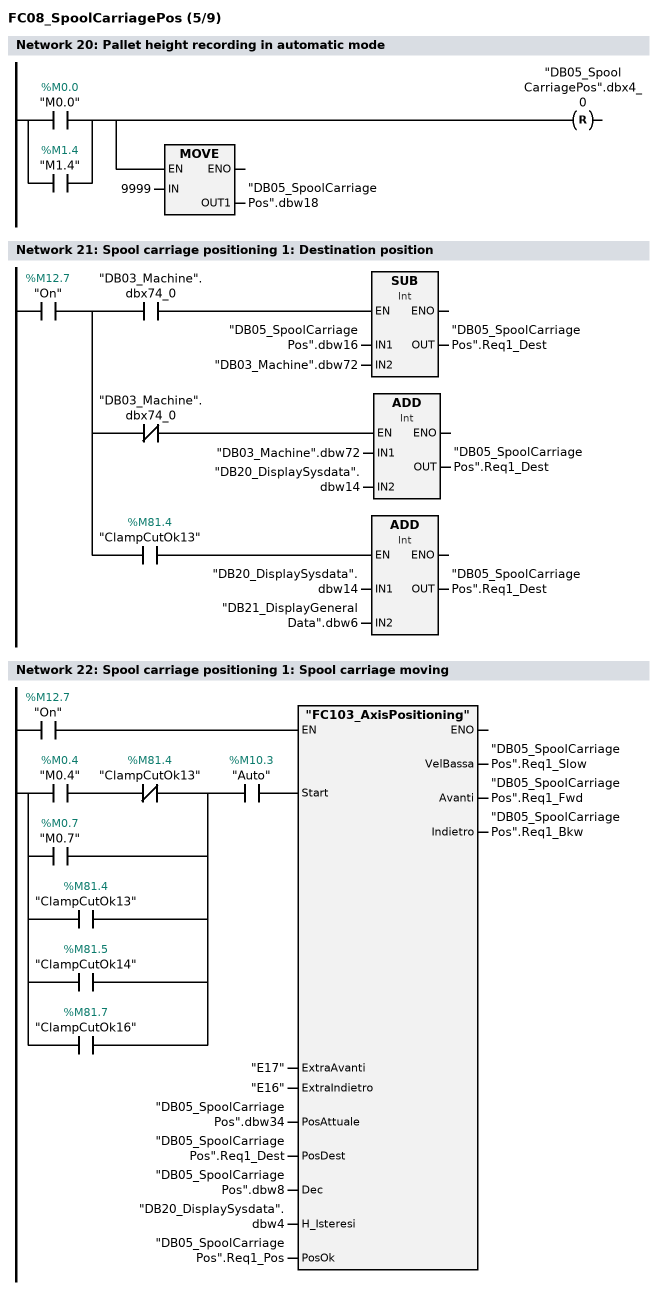
   RUNG wire#powerrail
      Contact( "M0.0" )
      wire#w1
      R_Coil( "DB05_SpoolCarriagePos".dbx4_0 )
   END_RUNG
   RUNG wire#powerrail
      Contact( "M1.4" )
   END_RUNG wire#w1
   RUNG wire#w1
      { S7_GenerateENO := "TRUE" } Move(in := 9999, out1 => "DB05_SpoolCarriagePos".dbw18)
   END_RUNG
   // the same network as SCL:
   IF "M0.0" OR "M1.4" THEN
       "DB05_SpoolCarriagePos".dbx4_0 := FALSE;
       "DB05_SpoolCarriagePos".dbw18 := 9999;
   END_IF;
END_REGION

REGION Network 21: Spool carriage positioning 1: Destination position
   RUNG wire#powerrail
      Contact( "On" )
      wire#w1
      Contact( "DB03_Machine".dbx74_0 )
      { S7_Templates := "SrcType := Int"; S7_GenerateENO := "TRUE" } Sub(in1 := "DB05_SpoolCarriagePos".dbw16, in2 := "DB03_Machine".dbw72, out => "DB05_SpoolCarriagePos".Req1_Dest)
   END_RUNG
   RUNG wire#w1
      I_Contact( "DB03_Machine".dbx74_0 )
      { S7_Templates := "SrcType := Int"; S7_GenerateENO := "TRUE" } Add(in1 := "DB03_Machine".dbw72, in2 := "DB20_DisplaySysdata".dbw14, out => "DB05_SpoolCarriagePos".Req1_Dest)
   END_RUNG
   RUNG wire#w1
      Contact( "ClampCutOk13" )
      { S7_Templates := "SrcType := Int"; S7_GenerateENO := "TRUE" } Add(in1 := "DB20_DisplaySysdata".dbw14, in2 := "DB21_DisplayGeneralData".dbw6, out => "DB05_SpoolCarriagePos".Req1_Dest)
   END_RUNG
   // the same network as SCL:
   IF "On" AND "DB03_Machine".dbx74_0 THEN
       "DB05_SpoolCarriagePos".Req1_Dest := "DB05_SpoolCarriagePos".dbw16 - "DB03_Machine".dbw72;
   END_IF;
   IF "On" AND NOT "DB03_Machine".dbx74_0 THEN
       "DB05_SpoolCarriagePos".Req1_Dest := "DB03_Machine".dbw72 + "DB20_DisplaySysdata".dbw14;
   END_IF;
   IF "On" AND "ClampCutOk13" THEN
       "DB05_SpoolCarriagePos".Req1_Dest := "DB20_DisplaySysdata".dbw14 + "DB21_DisplayGeneralData".dbw6;
   END_IF;
END_REGION

REGION Network 22: Spool carriage positioning 1: Spool carriage moving
   RUNG wire#powerrail
      Contact( "On" )
      "FC103_AxisPositioning"(Start := wire#w2, ExtraAvanti := "E17", ExtraIndietro := "E16", PosAttuale := "DB05_SpoolCarriagePos".dbw34, PosDest := "DB05_SpoolCarriagePos".Req1_Dest, Dec := "DB05_SpoolCarriagePos".dbw8, H_Isteresi := "DB20_DisplaySysdata".dbw4, PosOk := "DB05_SpoolCarriagePos".Req1_Pos, VelBassa => "DB05_SpoolCarriagePos".Req1_Slow, Avanti => "DB05_SpoolCarriagePos".Req1_Fwd, Indietro => "DB05_SpoolCarriagePos".Req1_Bkw)
   END_RUNG
   RUNG wire#powerrail
      Contact( "M0.4" )
      I_Contact( "ClampCutOk13" )
      wire#w1
      Contact( "Auto" )
   END_RUNG wire#w2
   RUNG wire#powerrail
      Contact( "M0.7" )
   END_RUNG wire#w1
   RUNG wire#powerrail
      Contact( "ClampCutOk13" )
   END_RUNG wire#w1
   RUNG wire#powerrail
      Contact( "ClampCutOk14" )
   END_RUNG wire#w1
   RUNG wire#powerrail
      Contact( "ClampCutOk16" )
   END_RUNG wire#w1
   // the same network as SCL:
   IF "On" THEN
       "FC103_AxisPositioning"(Start := (("M0.4" AND NOT "ClampCutOk13") OR "M0.7" OR "ClampCutOk13" OR "ClampCutOk14" OR "ClampCutOk16") AND "Auto",
                               ExtraAvanti := "E17",
                               ExtraIndietro := "E16",
                               PosAttuale := "DB05_SpoolCarriagePos".dbw34,
                               PosDest := "DB05_SpoolCarriagePos".Req1_Dest,
                               Dec := "DB05_SpoolCarriagePos".dbw8,
                               H_Isteresi := "DB20_DisplaySysdata".dbw4,
                               PosOk := "DB05_SpoolCarriagePos".Req1_Pos,
                               VelBassa => "DB05_SpoolCarriagePos".Req1_Slow,
                               Avanti => "DB05_SpoolCarriagePos".Req1_Fwd,
                               Indietro => "DB05_SpoolCarriagePos".Req1_Bkw);
   END_IF;
END_REGION

REGION Network 23: Spool carriage positioning 2: Destination position
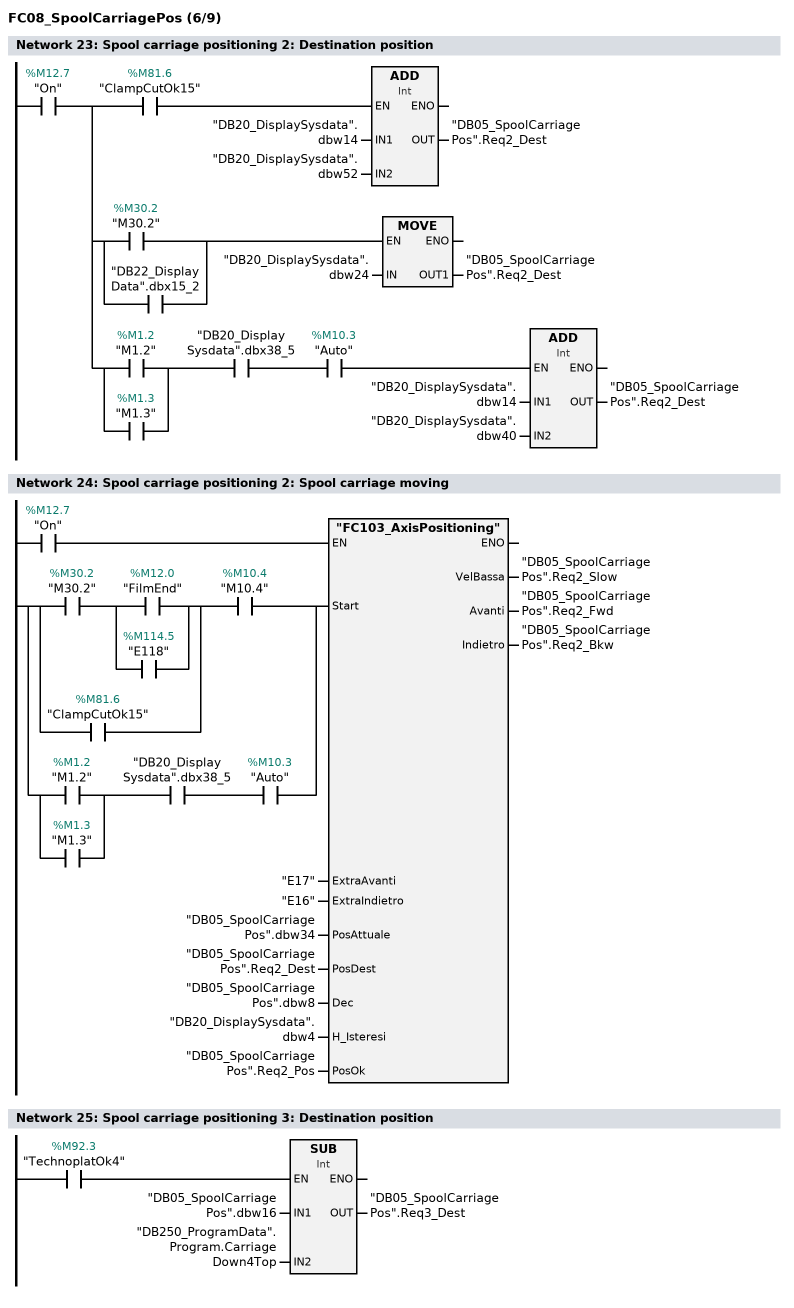
   RUNG wire#powerrail
      Contact( "On" )
      wire#w1
      Contact( "ClampCutOk15" )
      { S7_Templates := "SrcType := Int"; S7_GenerateENO := "TRUE" } Add(in1 := "DB20_DisplaySysdata".dbw14, in2 := "DB20_DisplaySysdata".dbw52, out => "DB05_SpoolCarriagePos".Req2_Dest)
   END_RUNG
   RUNG wire#w1
      Contact( "M30.2" )
      wire#w2
      { S7_GenerateENO := "TRUE" } Move(in := "DB20_DisplaySysdata".dbw24, out1 => "DB05_SpoolCarriagePos".Req2_Dest)
   END_RUNG
   RUNG wire#w1
      Contact( "DB22_DisplayData".dbx15_2 )
   END_RUNG wire#w2
   RUNG wire#w1
      Contact( "M1.2" )
      wire#w3
      Contact( "DB20_DisplaySysdata".dbx38_5 )
      Contact( "Auto" )
      { S7_Templates := "SrcType := Int"; S7_GenerateENO := "TRUE" } Add(in1 := "DB20_DisplaySysdata".dbw14, in2 := "DB20_DisplaySysdata".dbw40, out => "DB05_SpoolCarriagePos".Req2_Dest)
   END_RUNG
   RUNG wire#w1
      Contact( "M1.3" )
   END_RUNG wire#w3
   // the same network as SCL:
   IF "On" AND "ClampCutOk15" THEN
       "DB05_SpoolCarriagePos".Req2_Dest := "DB20_DisplaySysdata".dbw14 + "DB20_DisplaySysdata".dbw52;
   END_IF;
   IF "On" AND ("M30.2" OR "DB22_DisplayData".dbx15_2) THEN
       "DB05_SpoolCarriagePos".Req2_Dest := "DB20_DisplaySysdata".dbw24;
   END_IF;
   IF "On" AND ("M1.2" OR "M1.3") AND "DB20_DisplaySysdata".dbx38_5 AND "Auto" THEN
       "DB05_SpoolCarriagePos".Req2_Dest := "DB20_DisplaySysdata".dbw14 + "DB20_DisplaySysdata".dbw40;
   END_IF;
END_REGION

REGION Network 24: Spool carriage positioning 2: Spool carriage moving
   RUNG wire#powerrail
      Contact( "On" )
      "FC103_AxisPositioning"(Start := wire#w4, ExtraAvanti := "E17", ExtraIndietro := "E16", PosAttuale := "DB05_SpoolCarriagePos".dbw34, PosDest := "DB05_SpoolCarriagePos".Req2_Dest, Dec := "DB05_SpoolCarriagePos".dbw8, H_Isteresi := "DB20_DisplaySysdata".dbw4, PosOk := "DB05_SpoolCarriagePos".Req2_Pos, VelBassa => "DB05_SpoolCarriagePos".Req2_Slow, Avanti => "DB05_SpoolCarriagePos".Req2_Fwd, Indietro => "DB05_SpoolCarriagePos".Req2_Bkw)
   END_RUNG
   RUNG wire#powerrail
      Contact( "M30.2" )
      wire#w1
      Contact( "FilmEnd" )
      wire#w2
      Contact( "M10.4" )
   END_RUNG wire#w4
   RUNG wire#w1
      Contact( "E118" )
   END_RUNG wire#w2
   RUNG wire#powerrail
      Contact( "ClampCutOk15" )
   END_RUNG wire#w2
   RUNG wire#powerrail
      Contact( "M1.2" )
      wire#w3
      Contact( "DB20_DisplaySysdata".dbx38_5 )
      Contact( "Auto" )
   END_RUNG wire#w4
   RUNG wire#powerrail
      Contact( "M1.3" )
   END_RUNG wire#w3
   // the same network as SCL:
   IF "On" THEN
       "FC103_AxisPositioning"(Start := ((("M30.2" AND ("FilmEnd" OR "E118")) OR "ClampCutOk15") AND "M10.4") OR (("M1.2" OR "M1.3") AND "DB20_DisplaySysdata".dbx38_5 AND "Auto"),
                               ExtraAvanti := "E17",
                               ExtraIndietro := "E16",
                               PosAttuale := "DB05_SpoolCarriagePos".dbw34,
                               PosDest := "DB05_SpoolCarriagePos".Req2_Dest,
                               Dec := "DB05_SpoolCarriagePos".dbw8,
                               H_Isteresi := "DB20_DisplaySysdata".dbw4,
                               PosOk := "DB05_SpoolCarriagePos".Req2_Pos,
                               VelBassa => "DB05_SpoolCarriagePos".Req2_Slow,
                               Avanti => "DB05_SpoolCarriagePos".Req2_Fwd,
                               Indietro => "DB05_SpoolCarriagePos".Req2_Bkw);
   END_IF;
END_REGION

REGION Network 25: Spool carriage positioning 3: Destination position
   RUNG wire#powerrail
      Contact( "TechnoplatOk4" )
      { S7_Templates := "SrcType := Int"; S7_GenerateENO := "TRUE" } Sub(in1 := "DB05_SpoolCarriagePos".dbw16, in2 := "DB250_ProgramData".Program.CarriageDown4Top, out => "DB05_SpoolCarriagePos".Req3_Dest)
   END_RUNG
   // the same network as SCL:
   IF "TechnoplatOk4" THEN
       "DB05_SpoolCarriagePos".Req3_Dest := "DB05_SpoolCarriagePos".dbw16 - "DB250_ProgramData".Program.CarriageDown4Top;
   END_IF;
END_REGION

REGION Network 26: Spool carriage positioning 3: Spool carriage moving
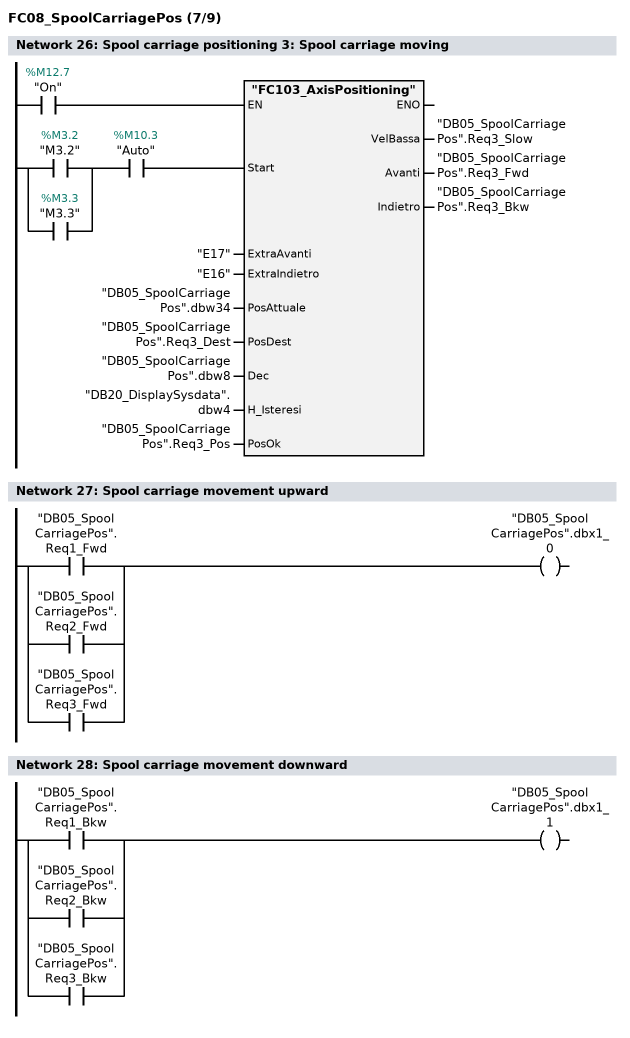
   RUNG wire#powerrail
      Contact( "On" )
      "FC103_AxisPositioning"(Start := wire#w2, ExtraAvanti := "E17", ExtraIndietro := "E16", PosAttuale := "DB05_SpoolCarriagePos".dbw34, PosDest := "DB05_SpoolCarriagePos".Req3_Dest, Dec := "DB05_SpoolCarriagePos".dbw8, H_Isteresi := "DB20_DisplaySysdata".dbw4, PosOk := "DB05_SpoolCarriagePos".Req3_Pos, VelBassa => "DB05_SpoolCarriagePos".Req3_Slow, Avanti => "DB05_SpoolCarriagePos".Req3_Fwd, Indietro => "DB05_SpoolCarriagePos".Req3_Bkw)
   END_RUNG
   RUNG wire#powerrail
      Contact( "M3.2" )
      wire#w1
      Contact( "Auto" )
   END_RUNG wire#w2
   RUNG wire#powerrail
      Contact( "M3.3" )
   END_RUNG wire#w1
   // the same network as SCL:
   IF "On" THEN
       "FC103_AxisPositioning"(Start := ("M3.2" OR "M3.3") AND "Auto",
                               ExtraAvanti := "E17",
                               ExtraIndietro := "E16",
                               PosAttuale := "DB05_SpoolCarriagePos".dbw34,
                               PosDest := "DB05_SpoolCarriagePos".Req3_Dest,
                               Dec := "DB05_SpoolCarriagePos".dbw8,
                               H_Isteresi := "DB20_DisplaySysdata".dbw4,
                               PosOk := "DB05_SpoolCarriagePos".Req3_Pos,
                               VelBassa => "DB05_SpoolCarriagePos".Req3_Slow,
                               Avanti => "DB05_SpoolCarriagePos".Req3_Fwd,
                               Indietro => "DB05_SpoolCarriagePos".Req3_Bkw);
   END_IF;
END_REGION

REGION Network 27: Spool carriage movement upward
   RUNG wire#powerrail
      Contact( "DB05_SpoolCarriagePos".Req1_Fwd )
      wire#w1
      Coil( "DB05_SpoolCarriagePos".dbx1_0 )
   END_RUNG
   RUNG wire#powerrail
      Contact( "DB05_SpoolCarriagePos".Req2_Fwd )
   END_RUNG wire#w1
   RUNG wire#powerrail
      Contact( "DB05_SpoolCarriagePos".Req3_Fwd )
   END_RUNG wire#w1
   // the same network as SCL:
   "DB05_SpoolCarriagePos".dbx1_0 := "DB05_SpoolCarriagePos".Req1_Fwd OR "DB05_SpoolCarriagePos".Req2_Fwd OR "DB05_SpoolCarriagePos".Req3_Fwd;
END_REGION

REGION Network 28: Spool carriage movement downward
   RUNG wire#powerrail
      Contact( "DB05_SpoolCarriagePos".Req1_Bkw )
      wire#w1
      Coil( "DB05_SpoolCarriagePos".dbx1_1 )
   END_RUNG
   RUNG wire#powerrail
      Contact( "DB05_SpoolCarriagePos".Req2_Bkw )
   END_RUNG wire#w1
   RUNG wire#powerrail
      Contact( "DB05_SpoolCarriagePos".Req3_Bkw )
   END_RUNG wire#w1
   // the same network as SCL:
   "DB05_SpoolCarriagePos".dbx1_1 := "DB05_SpoolCarriagePos".Req1_Bkw OR "DB05_SpoolCarriagePos".Req2_Bkw OR "DB05_SpoolCarriagePos".Req3_Bkw;
END_REGION

REGION Network 29: Spool carriage deceleration on carriage positioning
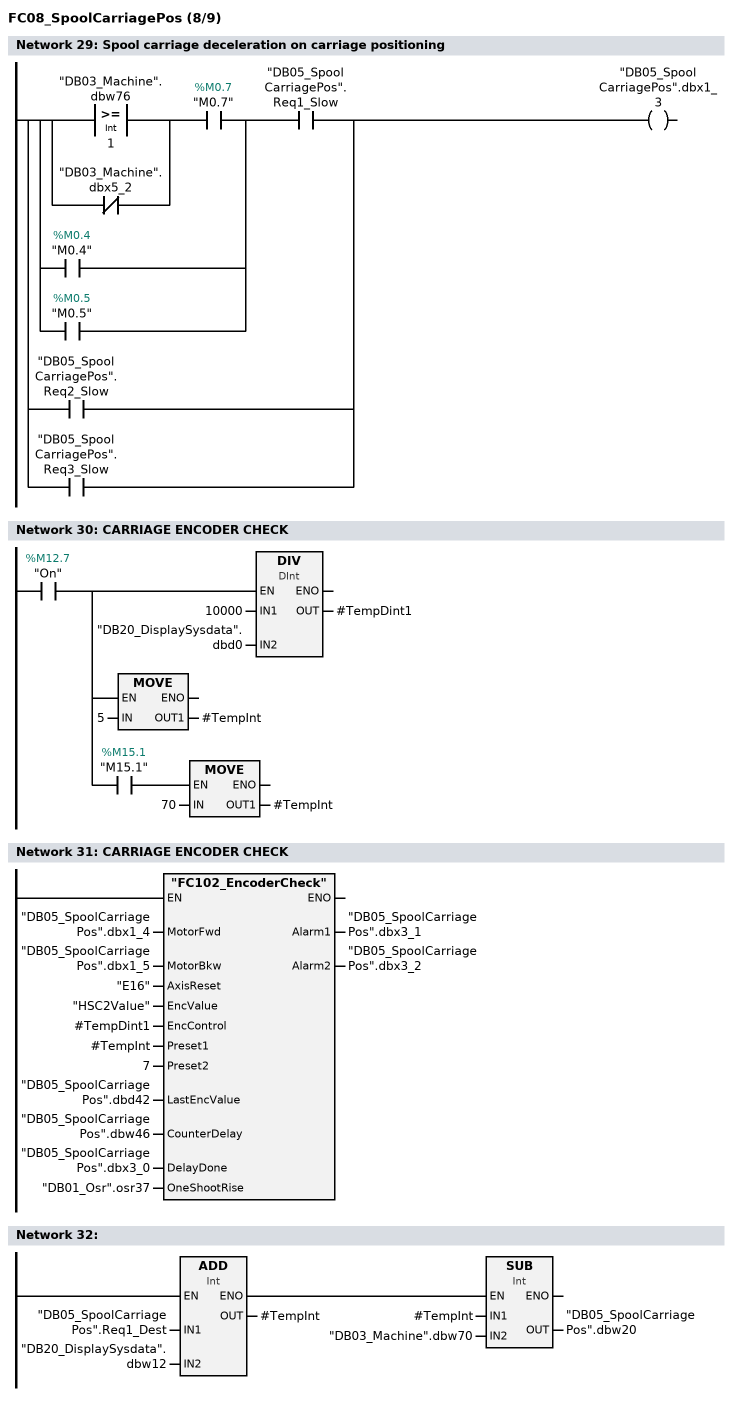
   RUNG wire#powerrail
      { S7_Templates := "SrcType := Int" } GE_Contact(in1 := "DB03_Machine".dbw76, in2 := 1)
      wire#w1
      Contact( "M0.7" )
      wire#w2
      Contact( "DB05_SpoolCarriagePos".Req1_Slow )
      wire#w3
      Coil( "DB05_SpoolCarriagePos".dbx1_3 )
   END_RUNG
   RUNG wire#powerrail
      I_Contact( "DB03_Machine".dbx5_2 )
   END_RUNG wire#w1
   RUNG wire#powerrail
      Contact( "M0.4" )
   END_RUNG wire#w2
   RUNG wire#powerrail
      Contact( "M0.5" )
   END_RUNG wire#w2
   RUNG wire#powerrail
      Contact( "DB05_SpoolCarriagePos".Req2_Slow )
   END_RUNG wire#w3
   RUNG wire#powerrail
      Contact( "DB05_SpoolCarriagePos".Req3_Slow )
   END_RUNG wire#w3
   // the same network as SCL:
   "DB05_SpoolCarriagePos".dbx1_3 := ((((("DB03_Machine".dbw76 >= 1) OR NOT "DB03_Machine".dbx5_2) AND "M0.7") OR "M0.4" OR "M0.5") AND "DB05_SpoolCarriagePos".Req1_Slow) OR "DB05_SpoolCarriagePos".Req2_Slow OR "DB05_SpoolCarriagePos".Req3_Slow;
END_REGION

REGION Network 30: CARRIAGE ENCODER CHECK
   RUNG wire#powerrail
      Contact( "On" )
      wire#w1
      { S7_Templates := "SrcType := DInt"; S7_GenerateENO := "TRUE" } Div(in1 := 10000, in2 := "DB20_DisplaySysdata".dbd0, out => #TempDint1)
   END_RUNG
   RUNG wire#w1
      { S7_GenerateENO := "TRUE" } Move(in := 5, out1 => #TempInt)
   END_RUNG
   RUNG wire#w1
      Contact( "M15.1" )
      { S7_GenerateENO := "TRUE" } Move(in := 70, out1 => #TempInt)
   END_RUNG
   // the same network as SCL:
   IF "On" THEN
       #TempDint1 := 10000 / "DB20_DisplaySysdata".dbd0;
       #TempInt := 5;
   END_IF;
   IF "On" AND "M15.1" THEN #TempInt := 70; END_IF;
END_REGION

REGION Network 31: CARRIAGE ENCODER CHECK
   RUNG wire#powerrail
      "FC102_EncoderCheck"(MotorFwd := "DB05_SpoolCarriagePos".dbx1_4, MotorBkw := "DB05_SpoolCarriagePos".dbx1_5, AxisReset := "E16", EncValue := "HSC2Value", EncControl := #TempDint1, Preset1 := #TempInt, Preset2 := 7, LastEncValue := "DB05_SpoolCarriagePos".dbd42, CounterDelay := "DB05_SpoolCarriagePos".dbw46, DelayDone := "DB05_SpoolCarriagePos".dbx3_0, OneShootRise := "DB01_Osr".osr37, Alarm1 => "DB05_SpoolCarriagePos".dbx3_1, Alarm2 => "DB05_SpoolCarriagePos".dbx3_2)
   END_RUNG
   // the same network as SCL:
   "FC102_EncoderCheck"(MotorFwd := "DB05_SpoolCarriagePos".dbx1_4,
                        MotorBkw := "DB05_SpoolCarriagePos".dbx1_5,
                        AxisReset := "E16",
                        EncValue := "HSC2Value",
                        EncControl := #TempDint1,
                        Preset1 := #TempInt,
                        Preset2 := 7,
                        LastEncValue := "DB05_SpoolCarriagePos".dbd42,
                        CounterDelay := "DB05_SpoolCarriagePos".dbw46,
                        DelayDone := "DB05_SpoolCarriagePos".dbx3_0,
                        OneShootRise := "DB01_Osr".osr37,
                        Alarm1 => "DB05_SpoolCarriagePos".dbx3_1,
                        Alarm2 => "DB05_SpoolCarriagePos".dbx3_2);
END_REGION

REGION Network 32
   RUNG wire#powerrail
      { S7_Templates := "SrcType := Int"; S7_GenerateENO := "TRUE" } Add(in1 := "DB05_SpoolCarriagePos".Req1_Dest, in2 := "DB20_DisplaySysdata".dbw12, out => #TempInt)
      { S7_Templates := "SrcType := Int"; S7_GenerateENO := "TRUE" } Sub(in1 := #TempInt, in2 := "DB03_Machine".dbw70, out => "DB05_SpoolCarriagePos".dbw20)
   END_RUNG
   // the same network as SCL:
   // ENO of a box is taken as its EN; it also drops when the box reports an error
   #TempInt := "DB05_SpoolCarriagePos".Req1_Dest + "DB20_DisplaySysdata".dbw12;
   "DB05_SpoolCarriagePos".dbw20 := #TempInt - "DB03_Machine".dbw70;
END_REGION

REGION Network 33
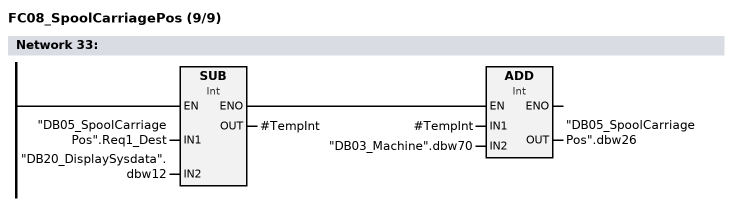
   RUNG wire#powerrail
      { S7_Templates := "SrcType := Int"; S7_GenerateENO := "TRUE" } Sub(in1 := "DB05_SpoolCarriagePos".Req1_Dest, in2 := "DB20_DisplaySysdata".dbw12, out => #TempInt)
      { S7_Templates := "SrcType := Int"; S7_GenerateENO := "TRUE" } Add(in1 := #TempInt, in2 := "DB03_Machine".dbw70, out => "DB05_SpoolCarriagePos".dbw26)
   END_RUNG
   // the same network as SCL:
   // ENO of a box is taken as its EN; it also drops when the box reports an error
   #TempInt := "DB05_SpoolCarriagePos".Req1_Dest - "DB20_DisplaySysdata".dbw12;
   "DB05_SpoolCarriagePos".dbw26 := #TempInt + "DB03_Machine".dbw70;
END_REGION
END_FUNCTION

FUNCTION "FC103_AxisPositioning" : Void   // FC103, LAD
TITLE = Axis positioning
{ S7_Optimized_Access := 'FALSE' }
AUTHOR : Robopac
VERSION : 0.0
// stored: AutoNumber false, IsIECCheckEnabled false, SetENOAutomatically false, UDAEnableTagReadback false
   VAR_INPUT
      Start : Bool;   // Start dell'asse
      ExtraAvanti : Bool;   // Sensore di extracorsa avanti
      ExtraIndietro : Bool;   // Sensore di extracorsa indietro
      PosAttuale : Int;   // Posizione attule dell'asse
      PosDest : Int;   // Posizione di destinazione dell'asse
      Dec : Int;   // Decelerazione
      H_Isteresi : Int;   // Isteresi
   END_VAR
   VAR_OUTPUT
      VelBassa : Bool;   // Asse all'interno dell'intervallo di decelerazione
      Avanti : Bool;   // Asse avanti
      Indietro : Bool;   // Asse indietro
   END_VAR
   VAR_IN_OUT
      PosOk : Bool;   // Asse in posizione
   END_VAR
   VAR_TEMP
      PosDestMenoH : Int;   // Posizione di destinazione asse-Isteresi
      PosDestPiuH : Int;   // Posizione di destinazione asse+Isteresi
      PosDestMenoDec : Int;   // Posizione di destinazione asse-Decelerazione
      PosDestPiuDec : Int;   // Posizione di destinazione asse+Decelerazione
   END_VAR
   VAR_TEMP   // added for the SCL form of the ladder/FBD networks
      _w1 : Bool;
   END_VAR
BEGIN

REGION Network 1
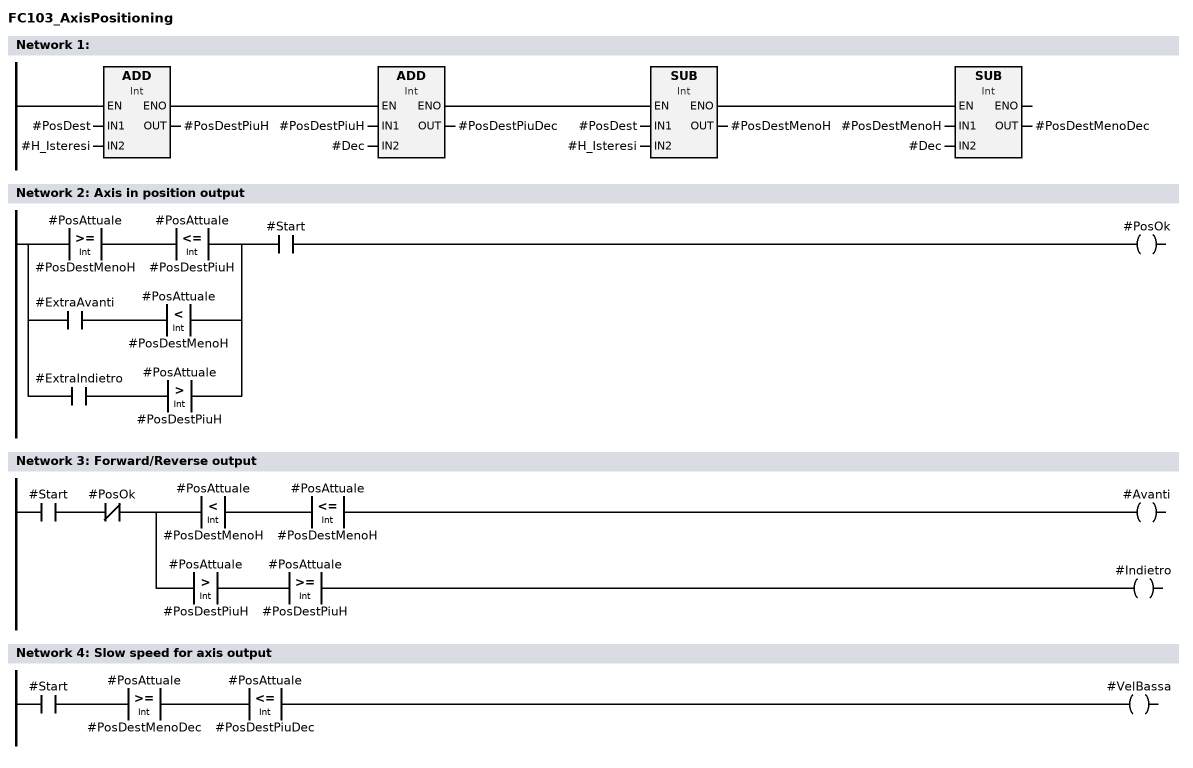
   RUNG wire#powerrail
      { S7_Templates := "SrcType := Int"; S7_GenerateENO := "TRUE" } Add(in1 := #PosDest, in2 := #H_Isteresi, out => #PosDestPiuH)
      { S7_Templates := "SrcType := Int"; S7_GenerateENO := "TRUE" } Add(in1 := #PosDestPiuH, in2 := #Dec, out => #PosDestPiuDec)
      { S7_Templates := "SrcType := Int"; S7_GenerateENO := "TRUE" } Sub(in1 := #PosDest, in2 := #H_Isteresi, out => #PosDestMenoH)
      { S7_Templates := "SrcType := Int"; S7_GenerateENO := "TRUE" } Sub(in1 := #PosDestMenoH, in2 := #Dec, out => #PosDestMenoDec)
   END_RUNG
   // the same network as SCL:
   // ENO of a box is taken as its EN; it also drops when the box reports an error
   #PosDestPiuH := #PosDest + #H_Isteresi;
   #PosDestPiuDec := #PosDestPiuH + #Dec;
   #PosDestMenoH := #PosDest - #H_Isteresi;
   #PosDestMenoDec := #PosDestMenoH - #Dec;
END_REGION

REGION Network 2: Axis in position output
   RUNG wire#powerrail
      { S7_Templates := "SrcType := Int" } GE_Contact(in1 := #PosAttuale, in2 := #PosDestMenoH)
      { S7_Templates := "SrcType := Int" } LE_Contact(in1 := #PosAttuale, in2 := #PosDestPiuH)
      wire#w1
      Contact( #Start )
      Coil( #PosOk )
   END_RUNG
   RUNG wire#powerrail
      Contact( #ExtraAvanti )
      { S7_Templates := "SrcType := Int" } LT_Contact(in1 := #PosAttuale, in2 := #PosDestMenoH)
   END_RUNG wire#w1
   RUNG wire#powerrail
      Contact( #ExtraIndietro )
      { S7_Templates := "SrcType := Int" } GT_Contact(in1 := #PosAttuale, in2 := #PosDestPiuH)
   END_RUNG wire#w1
   // the same network as SCL:
   #PosOk := (((#PosAttuale >= #PosDestMenoH) AND (#PosAttuale <= #PosDestPiuH)) OR (#ExtraAvanti AND (#PosAttuale < #PosDestMenoH)) OR (#ExtraIndietro AND (#PosAttuale > #PosDestPiuH))) AND #Start;
END_REGION

REGION Network 3: Forward/Reverse output
   RUNG wire#powerrail
      Contact( #Start )
      I_Contact( #PosOk )
      wire#w1
      { S7_Templates := "SrcType := Int" } LT_Contact(in1 := #PosAttuale, in2 := #PosDestMenoH)
      { S7_Templates := "SrcType := Int" } LE_Contact(in1 := #PosAttuale, in2 := #PosDestMenoH)
      Coil( #Avanti )
   END_RUNG
   RUNG wire#w1
      { S7_Templates := "SrcType := Int" } GT_Contact(in1 := #PosAttuale, in2 := #PosDestPiuH)
      { S7_Templates := "SrcType := Int" } GE_Contact(in1 := #PosAttuale, in2 := #PosDestPiuH)
      Coil( #Indietro )
   END_RUNG
   // the same network as SCL:
   #_w1 := #Start AND NOT #PosOk;
   #Avanti := #_w1 AND (#PosAttuale < #PosDestMenoH) AND (#PosAttuale <= #PosDestMenoH);
   #Indietro := #_w1 AND (#PosAttuale > #PosDestPiuH) AND (#PosAttuale >= #PosDestPiuH);
END_REGION

REGION Network 4: Slow speed for axis output
   RUNG wire#powerrail
      Contact( #Start )
      { S7_Templates := "SrcType := Int" } GE_Contact(in1 := #PosAttuale, in2 := #PosDestMenoDec)
      { S7_Templates := "SrcType := Int" } LE_Contact(in1 := #PosAttuale, in2 := #PosDestPiuDec)
      Coil( #VelBassa )
   END_RUNG
   // the same network as SCL:
   #VelBassa := #Start AND (#PosAttuale >= #PosDestMenoDec) AND (#PosAttuale <= #PosDestPiuDec);
END_REGION
END_FUNCTION

FUNCTION "FC102_EncoderCheck" : Void   // FC102, LAD
{ S7_Optimized_Access := 'FALSE' }
AUTHOR : AetnaG
VERSION : 0.0
// stored: AutoNumber false, IsIECCheckEnabled false, SetENOAutomatically false, UDAEnableTagReadback false
   VAR_INPUT
      MotorFwd : Bool;
      MotorBkw : Bool;
      AxisReset : Bool;
      EncValue : DInt;
      EncControl : DInt;
      Preset1 : Int;
      Preset2 : Int;
   END_VAR
   VAR_OUTPUT
      Alarm1 : Bool;
      Alarm2 : Bool;
   END_VAR
   VAR_IN_OUT
      LastEncValue : DInt;
      CounterDelay : Int;
      DelayDone : Bool;
      OneShootRise : Bool;
   END_VAR
   VAR_TEMP
      EncDifference : DInt;
      EncControlOpp : DInt;
      CounterReset : Bool;
   END_VAR
   VAR_TEMP   // added for the SCL form of the ladder/FBD networks
      _w1 : Bool;
   END_VAR
BEGIN

REGION Network 1
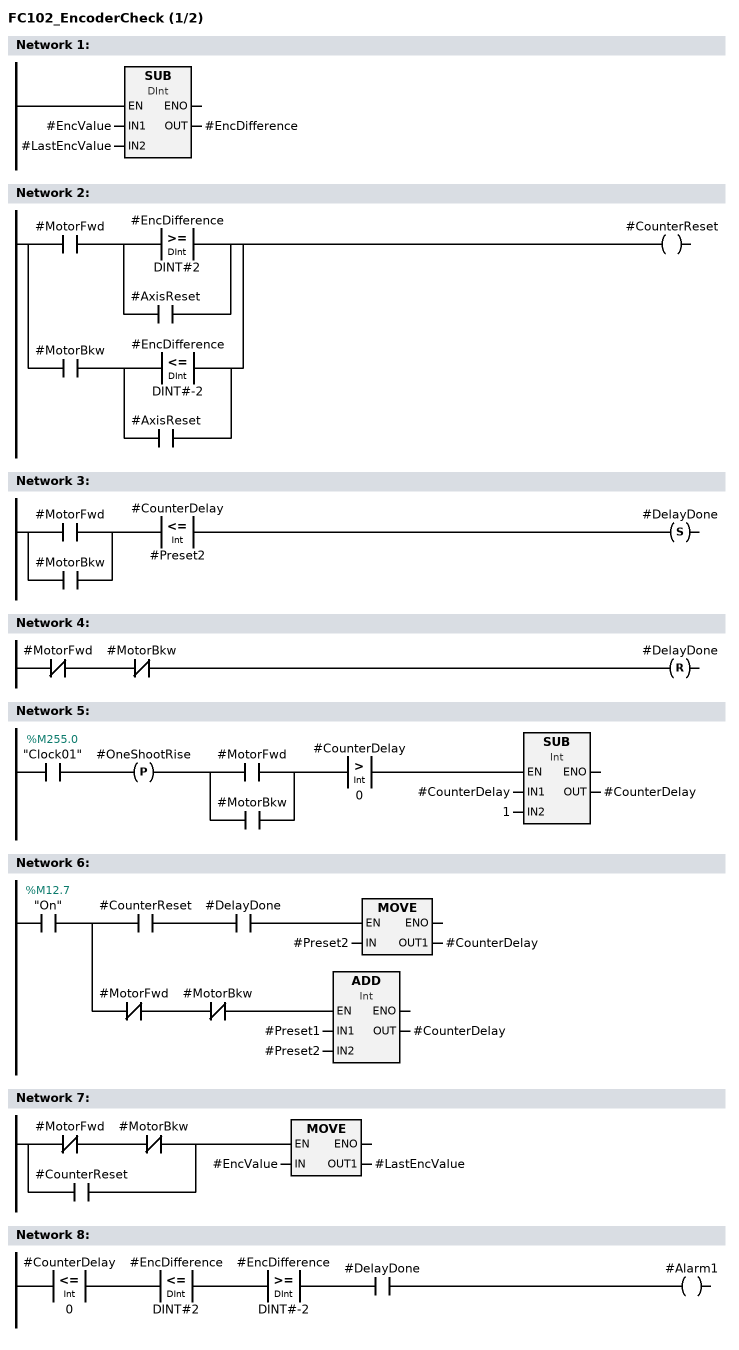
   RUNG wire#powerrail
      { S7_Templates := "SrcType := DInt"; S7_GenerateENO := "TRUE" } Sub(in1 := #EncValue, in2 := #LastEncValue, out => #EncDifference)
   END_RUNG
   // the same network as SCL:
   #EncDifference := #EncValue - #LastEncValue;
END_REGION

REGION Network 2
   RUNG wire#powerrail
      Contact( #MotorFwd )
      wire#w1
      { S7_Templates := "SrcType := DInt" } GE_Contact(in1 := #EncDifference, in2 := DINT#2)
      wire#w2
      Coil( #CounterReset )
   END_RUNG
   RUNG wire#w1
      Contact( #AxisReset )
   END_RUNG wire#w2
   RUNG wire#powerrail
      Contact( #MotorBkw )
      wire#w3
      { S7_Templates := "SrcType := DInt" } LE_Contact(in1 := #EncDifference, in2 := DINT#-2)
   END_RUNG wire#w2
   RUNG wire#w3
      Contact( #AxisReset )
   END_RUNG wire#w2
   // the same network as SCL:
   #CounterReset := (#MotorFwd AND ((#EncDifference >= DINT#2) OR #AxisReset)) OR (#MotorBkw AND ((#EncDifference <= DINT#-2) OR #AxisReset));
END_REGION

REGION Network 3
   RUNG wire#powerrail
      Contact( #MotorFwd )
      wire#w1
      { S7_Templates := "SrcType := Int" } LE_Contact(in1 := #CounterDelay, in2 := #Preset2)
      S_Coil( #DelayDone )
   END_RUNG
   RUNG wire#powerrail
      Contact( #MotorBkw )
   END_RUNG wire#w1
   // the same network as SCL:
   IF (#MotorFwd OR #MotorBkw) AND (#CounterDelay <= #Preset2) THEN #DelayDone := TRUE; END_IF;
END_REGION

REGION Network 4
   RUNG wire#powerrail
      I_Contact( #MotorFwd )
      I_Contact( #MotorBkw )
      R_Coil( #DelayDone )
   END_RUNG
   // the same network as SCL:
   IF NOT #MotorFwd AND NOT #MotorBkw THEN #DelayDone := FALSE; END_IF;
END_REGION

REGION Network 5
   RUNG wire#powerrail
      Contact( "Clock01" )
      P_Trig( #OneShootRise )
      wire#w1
      Contact( #MotorFwd )
      wire#w2
      { S7_Templates := "SrcType := Int" } GT_Contact(in1 := #CounterDelay, in2 := 0)
      { S7_Templates := "SrcType := Int"; S7_GenerateENO := "TRUE" } Sub(in1 := #CounterDelay, in2 := 1, out => #CounterDelay)
   END_RUNG
   RUNG wire#w1
      Contact( #MotorBkw )
   END_RUNG wire#w2
   // the same network as SCL:
   #_w1 := "Clock01" AND NOT #OneShootRise;   // rising edge
   #OneShootRise := "Clock01";
   IF #_w1 AND (#MotorFwd OR #MotorBkw) AND (#CounterDelay > 0) THEN
       #CounterDelay := #CounterDelay - 1;
   END_IF;
END_REGION

REGION Network 6
   RUNG wire#powerrail
      Contact( "On" )
      wire#w1
      Contact( #CounterReset )
      Contact( #DelayDone )
      { S7_GenerateENO := "TRUE" } Move(in := #Preset2, out1 => #CounterDelay)
   END_RUNG
   RUNG wire#w1
      I_Contact( #MotorFwd )
      I_Contact( #MotorBkw )
      { S7_Templates := "SrcType := Int"; S7_GenerateENO := "TRUE" } Add(in1 := #Preset1, in2 := #Preset2, out => #CounterDelay)
   END_RUNG
   // the same network as SCL:
   IF "On" AND #CounterReset AND #DelayDone THEN #CounterDelay := #Preset2; END_IF;
   IF "On" AND NOT #MotorFwd AND NOT #MotorBkw THEN #CounterDelay := #Preset1 + #Preset2; END_IF;
END_REGION

REGION Network 7
   RUNG wire#powerrail
      I_Contact( #MotorFwd )
      I_Contact( #MotorBkw )
      wire#w1
      { S7_GenerateENO := "TRUE" } Move(in := #EncValue, out1 => #LastEncValue)
   END_RUNG
   RUNG wire#powerrail
      Contact( #CounterReset )
   END_RUNG wire#w1
   // the same network as SCL:
   IF (NOT #MotorFwd AND NOT #MotorBkw) OR #CounterReset THEN #LastEncValue := #EncValue; END_IF;
END_REGION

REGION Network 8
   RUNG wire#powerrail
      { S7_Templates := "SrcType := Int" } LE_Contact(in1 := #CounterDelay, in2 := 0)
      { S7_Templates := "SrcType := DInt" } LE_Contact(in1 := #EncDifference, in2 := DINT#2)
      { S7_Templates := "SrcType := DInt" } GE_Contact(in1 := #EncDifference, in2 := DINT#-2)
      Contact( #DelayDone )
      Coil( #Alarm1 )
   END_RUNG
   // the same network as SCL:
   #Alarm1 := (#CounterDelay <= 0) AND (#EncDifference <= DINT#2) AND (#EncDifference >= DINT#-2) AND #DelayDone;
END_REGION

REGION Network 9
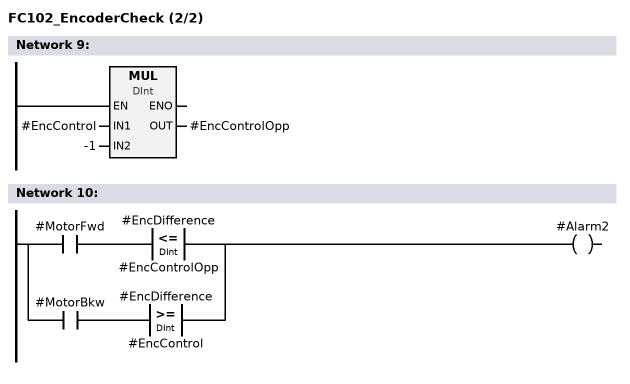
   RUNG wire#powerrail
      { S7_Templates := "SrcType := DInt"; S7_GenerateENO := "TRUE" } Mul(in1 := #EncControl, in2 := -1, out => #EncControlOpp)
   END_RUNG
   // the same network as SCL:
   #EncControlOpp := #EncControl * (-1);
END_REGION

REGION Network 10
   RUNG wire#powerrail
      Contact( #MotorFwd )
      { S7_Templates := "SrcType := DInt" } LE_Contact(in1 := #EncDifference, in2 := #EncControlOpp)
      wire#w1
      Coil( #Alarm2 )
   END_RUNG
   RUNG wire#powerrail
      Contact( #MotorBkw )
      { S7_Templates := "SrcType := DInt" } GE_Contact(in1 := #EncDifference, in2 := #EncControl)
   END_RUNG wire#w1
   // the same network as SCL:
   #Alarm2 := (#MotorFwd AND (#EncDifference <= #EncControlOpp)) OR (#MotorBkw AND (#EncDifference >= #EncControl));
END_REGION
END_FUNCTION

FUNCTION "FC58_TableRotationPos" : Void   // FC58, LAD
{ S7_Optimized_Access := 'FALSE' }
VERSION : 0.1
// stored: AutoNumber false, IsIECCheckEnabled false, SetENOAutomatically false, UDAEnableTagReadback false
   VAR_INPUT
      PHASE : Bool;
   END_VAR
   VAR_TEMP
      TempDInt3 : DInt;
      PulseOffset : DInt;
      AC1 : Real;
      AC2 : Real;
      AC3 : Real;
      DeltaV : Real;
      DeltaVMax : Real;
      VattpiuVmin : Real;
      VmaxpiuVmin : Real;
      AC1_INT : Int;
      PulseReset : Bool;
      TEMPOMAX : Real;
      TEMPO : Real;
      Encoder : Int;
      TempDint : DInt;
      TempInt : Int;
      TempDint2 : DInt;
      TempDInt4 : DInt;
      TempWord : Word;
   END_VAR
   VAR_TEMP   // added for the SCL form of the ladder/FBD networks
      _w1 : Bool;
   END_VAR
BEGIN

REGION Network 1
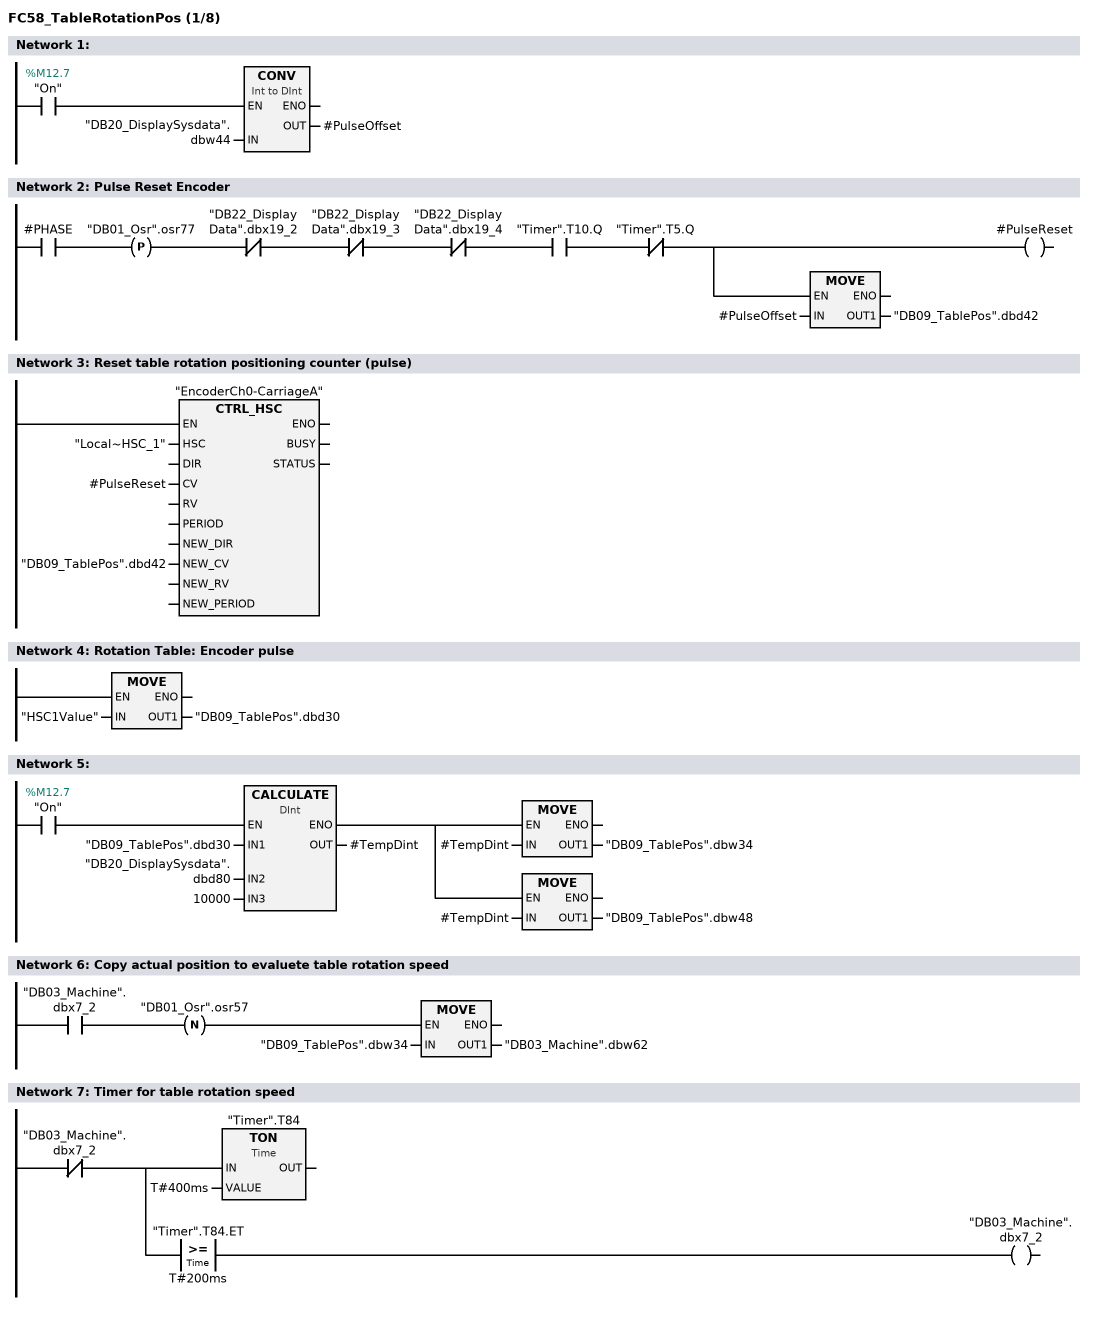
   RUNG wire#powerrail
      Contact( "On" )
      { S7_Templates := "[SrcType := Int, DestType := DInt]"; S7_GenerateENO := "TRUE" } Convert(in := "DB20_DisplaySysdata".dbw44, out => #PulseOffset)
   END_RUNG
   // the same network as SCL:
   IF "On" THEN #PulseOffset := INT_TO_DINT("DB20_DisplaySysdata".dbw44); END_IF;
END_REGION

REGION Network 2: Pulse Reset Encoder
   RUNG wire#powerrail
      Contact( #PHASE )
      P_Trig( "DB01_Osr".osr77 )
      I_Contact( "DB22_DisplayData".dbx19_2 )
      I_Contact( "DB22_DisplayData".dbx19_3 )
      I_Contact( "DB22_DisplayData".dbx19_4 )
      Contact( "Timer".T10.Q )
      I_Contact( "Timer".T5.Q )
      wire#w1
      Coil( #PulseReset )
   END_RUNG
   RUNG wire#w1
      { S7_GenerateENO := "TRUE" } Move(in := #PulseOffset, out1 => "DB09_TablePos".dbd42)
   END_RUNG
   // the same network as SCL:
   #_w1 := #PHASE AND NOT "DB01_Osr".osr77;   // rising edge
   "DB01_Osr".osr77 := #PHASE;
   #PulseReset := #_w1 AND NOT "DB22_DisplayData".dbx19_2 AND NOT "DB22_DisplayData".dbx19_3 AND NOT "DB22_DisplayData".dbx19_4 AND "Timer".T10.Q AND NOT "Timer".T5.Q;
   IF #PulseReset THEN "DB09_TablePos".dbd42 := #PulseOffset; END_IF;
END_REGION

REGION Network 3: Reset table rotation positioning counter (pulse)
   RUNG wire#powerrail
      "EncoderCh0-CarriageA".CTRL_HSC(HSC := "Local~HSC_1", DIR :=, CV := #PulseReset, RV :=, PERIOD :=, NEW_DIR :=, NEW_CV := "DB09_TablePos".dbd42, NEW_RV :=, NEW_PERIOD :=, BUSY =>, STATUS =>)
   END_RUNG
   // the same network as SCL:
   "EncoderCh0-CarriageA"(HSC := "Local~HSC_1", CV := #PulseReset, NEW_CV := "DB09_TablePos".dbd42);   // CTRL_HSC
END_REGION

REGION Network 4: Rotation Table: Encoder pulse
   RUNG wire#powerrail
      { S7_GenerateENO := "TRUE" } Move(in := "HSC1Value", out1 => "DB09_TablePos".dbd30)
   END_RUNG
   // the same network as SCL:
   "DB09_TablePos".dbd30 := "HSC1Value";
END_REGION

REGION Network 5
   RUNG wire#powerrail
      Contact( "On" )
      { S7_Templates := "SrcType := DInt"; S7_GenerateENO := "TRUE"; S7_Expression := "((In1*In2)/In3)" } Calculate(in1 := "DB09_TablePos".dbd30, in2 := "DB20_DisplaySysdata".dbd80, in3 := 10000, out => #TempDint)
      wire#w1
      { S7_GenerateENO := "TRUE" } Move(in := #TempDint, out1 => "DB09_TablePos".dbw34)
   END_RUNG
   RUNG wire#w1
      { S7_GenerateENO := "TRUE" } Move(in := #TempDint, out1 => "DB09_TablePos".dbw48)
   END_RUNG
   // the same network as SCL:
   // ENO of a box is taken as its EN; it also drops when the box reports an error
   IF "On" THEN
       #TempDint := (("DB09_TablePos".dbd30*"DB20_DisplaySysdata".dbd80)/10000);
       "DB09_TablePos".dbw34 := #TempDint;
       "DB09_TablePos".dbw48 := #TempDint;
   END_IF;
END_REGION

REGION Network 6: Copy actual position to evaluete table rotation speed
   RUNG wire#powerrail
      Contact( "DB03_Machine".dbx7_2 )
      N_Trig( "DB01_Osr".osr57 )
      { S7_GenerateENO := "TRUE" } Move(in := "DB09_TablePos".dbw34, out1 => "DB03_Machine".dbw62)
   END_RUNG
   // the same network as SCL:
   #_w1 := NOT "DB03_Machine".dbx7_2 AND "DB01_Osr".osr57;   // falling edge
   "DB01_Osr".osr57 := "DB03_Machine".dbx7_2;
   IF #_w1 THEN "DB03_Machine".dbw62 := "DB09_TablePos".dbw34; END_IF;
END_REGION

REGION Network 7: Timer for table rotation speed
   #_w1 := NOT "DB03_Machine".dbx7_2;
   "Timer".T84.TON(IN := #_w1, PT := T#400ms);   // TON coil
   "DB03_Machine".dbx7_2 := #_w1 AND ("Timer".T84.ET >= T#200ms);
END_REGION

REGION Network 8: Speed calculation (1)
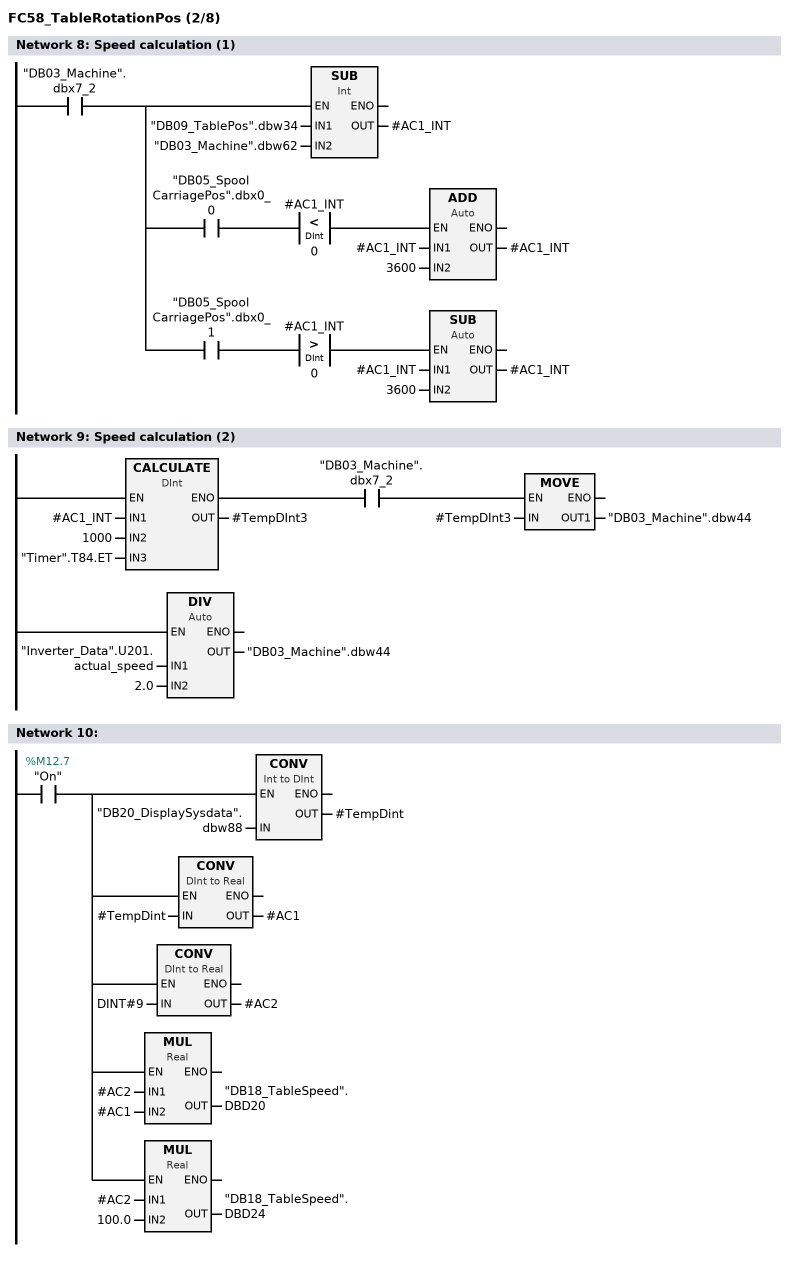
   RUNG wire#powerrail
      Contact( "DB03_Machine".dbx7_2 )
      wire#w1
      { S7_Templates := "SrcType := Int"; S7_GenerateENO := "TRUE" } Sub(in1 := "DB09_TablePos".dbw34, in2 := "DB03_Machine".dbw62, out => #AC1_INT)
   END_RUNG
   RUNG wire#w1
      Contact( "DB05_SpoolCarriagePos".dbx0_0 )
      { S7_Templates := "SrcType := DInt" } LT_Contact(in1 := #AC1_INT, in2 := 0)
      { S7_GenerateENO := "TRUE" } Add(in1 := #AC1_INT, in2 := 3600, out => #AC1_INT)
   END_RUNG
   RUNG wire#w1
      Contact( "DB05_SpoolCarriagePos".dbx0_1 )
      { S7_Templates := "SrcType := DInt" } GT_Contact(in1 := #AC1_INT, in2 := 0)
      { S7_GenerateENO := "TRUE" } Sub(in1 := #AC1_INT, in2 := 3600, out => #AC1_INT)
   END_RUNG
   // the same network as SCL:
   IF "DB03_Machine".dbx7_2 THEN #AC1_INT := "DB09_TablePos".dbw34 - "DB03_Machine".dbw62; END_IF;
   IF "DB03_Machine".dbx7_2 AND "DB05_SpoolCarriagePos".dbx0_0 AND (#AC1_INT < 0) THEN
       #AC1_INT := #AC1_INT + 3600;
   END_IF;
   IF "DB03_Machine".dbx7_2 AND "DB05_SpoolCarriagePos".dbx0_1 AND (#AC1_INT > 0) THEN
       #AC1_INT := #AC1_INT - 3600;
   END_IF;
END_REGION

REGION Network 9: Speed calculation (2)
   RUNG wire#powerrail
      { S7_Templates := "SrcType := DInt"; S7_GenerateENO := "TRUE"; S7_Expression := "((In1*In2)/In3)" } Calculate(in1 := #AC1_INT, in2 := 1000, in3 := "Timer".T84.ET, out => #TempDInt3)
      Contact( "DB03_Machine".dbx7_2 )
      { S7_GenerateENO := "TRUE" } Move(in := #TempDInt3, out1 => "DB03_Machine".dbw44)
   END_RUNG
   RUNG wire#powerrail
      Div(in1 := "Inverter_Data".U201.actual_speed, in2 := 2.0, out => "DB03_Machine".dbw44)
   END_RUNG
   // the same network as SCL:
   // ENO of a box is taken as its EN; it also drops when the box reports an error
   #TempDInt3 := ((#AC1_INT*1000)/"Timer".T84.ET);
   IF "DB03_Machine".dbx7_2 THEN "DB03_Machine".dbw44 := #TempDInt3; END_IF;
   "DB03_Machine".dbw44 := "Inverter_Data".U201.actual_speed / 2.0;
END_REGION

REGION Network 10
   RUNG wire#powerrail
      Contact( "On" )
      wire#w1
      { S7_Templates := "[SrcType := Int, DestType := DInt]"; S7_GenerateENO := "TRUE" } Convert(in := "DB20_DisplaySysdata".dbw88, out => #TempDint)
   END_RUNG
   RUNG wire#w1
      { S7_Templates := "[SrcType := DInt, DestType := Real]"; S7_GenerateENO := "TRUE" } Convert(in := #TempDint, out => #AC1)
   END_RUNG
   RUNG wire#w1
      { S7_Templates := "[SrcType := DInt, DestType := Real]"; S7_GenerateENO := "TRUE" } Convert(in := DINT#9, out => #AC2)
   END_RUNG
   RUNG wire#w1
      { S7_Templates := "SrcType := Real"; S7_GenerateENO := "TRUE" } Mul(in1 := #AC2, in2 := #AC1, out => "DB18_TableSpeed".DBD20)
   END_RUNG
   RUNG wire#w1
      { S7_Templates := "SrcType := Real"; S7_GenerateENO := "TRUE" } Mul(in1 := #AC2, in2 := 100.0, out => "DB18_TableSpeed".DBD24)
   END_RUNG
   // the same network as SCL:
   IF "On" THEN
       #TempDint := INT_TO_DINT("DB20_DisplaySysdata".dbw88);
       #AC1 := DINT_TO_REAL(#TempDint);
       #AC2 := DINT_TO_REAL(DINT#9);
       "DB18_TableSpeed".DBD20 := #AC2 * #AC1;
       "DB18_TableSpeed".DBD24 := #AC2 * 100.0;
   END_IF;
END_REGION

REGION Network 11
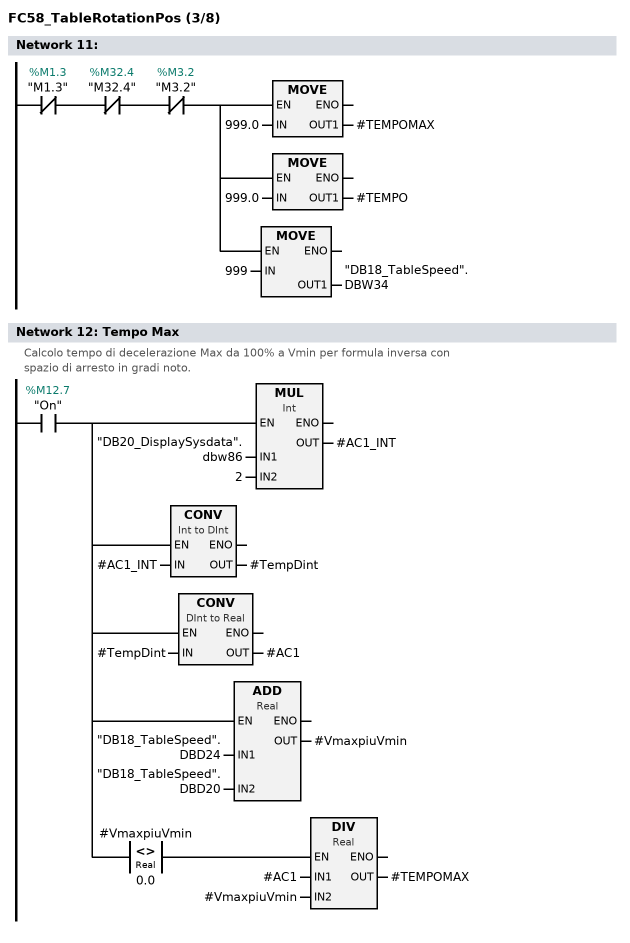
   RUNG wire#powerrail
      I_Contact( "M1.3" )
      I_Contact( "M32.4" )
      I_Contact( "M3.2" )
      wire#w1
      { S7_GenerateENO := "TRUE" } Move(in := 999.0, out1 => #TEMPOMAX)
   END_RUNG
   RUNG wire#w1
      { S7_GenerateENO := "TRUE" } Move(in := 999.0, out1 => #TEMPO)
   END_RUNG
   RUNG wire#w1
      { S7_GenerateENO := "TRUE" } Move(in := 999, out1 => "DB18_TableSpeed".DBW34)
   END_RUNG
   // the same network as SCL:
   IF NOT "M1.3" AND NOT "M32.4" AND NOT "M3.2" THEN
       #TEMPOMAX := 999.0;
       #TEMPO := 999.0;
       "DB18_TableSpeed".DBW34 := 999;
   END_IF;
END_REGION

REGION Network 12: Tempo Max
   // Calcolo tempo di decelerazione Max da 100% a Vmin per formula inversa con 
   // spazio di arresto in gradi noto.
   RUNG wire#powerrail
      Contact( "On" )
      wire#w1
      { S7_Templates := "SrcType := Int"; S7_GenerateENO := "TRUE" } Mul(in1 := "DB20_DisplaySysdata".dbw86, in2 := 2, out => #AC1_INT)
   END_RUNG
   RUNG wire#w1
      { S7_Templates := "[SrcType := Int, DestType := DInt]"; S7_GenerateENO := "TRUE" } Convert(in := #AC1_INT, out => #TempDint)
   END_RUNG
   RUNG wire#w1
      { S7_Templates := "[SrcType := DInt, DestType := Real]"; S7_GenerateENO := "TRUE" } Convert(in := #TempDint, out => #AC1)
   END_RUNG
   RUNG wire#w1
      { S7_Templates := "SrcType := Real"; S7_GenerateENO := "TRUE" } Add(in1 := "DB18_TableSpeed".DBD24, in2 := "DB18_TableSpeed".DBD20, out => #VmaxpiuVmin)
   END_RUNG
   RUNG wire#w1
      { S7_Templates := "SrcType := Real" } NE_Contact(in1 := #VmaxpiuVmin, in2 := 0.0)
      { S7_Templates := "SrcType := Real"; S7_GenerateENO := "TRUE" } Div(in1 := #AC1, in2 := #VmaxpiuVmin, out => #TEMPOMAX)
   END_RUNG
   // the same network as SCL:
   IF "On" THEN
       #AC1_INT := "DB20_DisplaySysdata".dbw86 * 2;
       #TempDint := INT_TO_DINT(#AC1_INT);
       #AC1 := DINT_TO_REAL(#TempDint);
       #VmaxpiuVmin := "DB18_TableSpeed".DBD24 + "DB18_TableSpeed".DBD20;
   END_IF;
   IF "On" AND (#VmaxpiuVmin <> 0.0) THEN #TEMPOMAX := #AC1 / #VmaxpiuVmin; END_IF;
END_REGION

REGION Network 13: Calcolo tempo di decelerazione da Vatt a Vmin per calcolo spazio di arresto
